  MoveL (T17595) to (111.78, 115.61, 18.9) mm, rotated rx 180 ry 0 rz -180 deg; joints [2.068, 71.073, -37.56, 3.741, -33.569, -3.119]
  Call Extruder 0.01417
  MoveL (T17596) to (111.39, 115.99, 18.9) mm, rotated rx 180 ry 0 rz -180 deg; joints [2.068, 71.073, -37.56, 3.741, -33.569, -3.119]
  Call Extruder 0.01304
  MoveL (T17597) to (110.9, 115.99, 18.9) mm, rotated rx 180 ry 0 rz -180 deg; joints [2.068, 71.073, -37.56, 3.741, -33.569, -3.119]
  Call Extruder 0.02638
  MoveL (T17598) to (111.61, 115.28, 18.9) mm, rotated rx 180 ry 0 rz -180 deg; joints [1.852, 70.394, -36.284, 3.299, -34.154, -2.731]
  Call Extruder 0.00969
  MoveL (T17599) to (111.44, 114.95, 18.9) mm, rotated rx 180 ry 0 rz -180 deg; joints [1.852, 70.394, -36.284, 3.299, -34.154, -2.731]
  Call Extruder 0.03859
  MoveL (T17600) to (110.4, 115.99, 18.9) mm, rotated rx 180 ry 0 rz -180 deg; joints [1.883, 70.309, -36.124, 3.349, -34.23, -2.77]
  Call Extruder 0.01304
  MoveL (T17601) to (109.91, 115.99, 18.9) mm, rotated rx 180 ry 0 rz -180 deg; joints [1.883, 70.309, -36.124, 3.349, -34.23, -2.77]
  Call Extruder 0.0508
  MoveL (T17602) to (111.27, 114.62, 18.9) mm, rotated rx 180 ry 0 rz -180 deg; joints [1.883, 70.309, -36.124, 3.349, -34.23, -2.77]
  Call Extruder 0.00969
  MoveL (T17603) to (111.11, 114.3, 18.9) mm, rotated rx 180 ry 0 rz -180 deg; joints [2.129, 71.08, -37.573, 3.852, -33.567, -3.211]
  Call Extruder 0.06301
  MoveL (T17604) to (109.41, 115.99, 18.9) mm, rotated rx 180 ry 0 rz -180 deg; joints [2.129, 71.08, -37.573, 3.852, -33.567, -3.211]
  Call Extruder 0.01304
  MoveL (T17605) to (108.91, 115.99, 18.9) mm, rotated rx 180 ry 0 rz -180 deg; joints [2.129, 71.08, -37.573, 3.852, -33.567, -3.211]
  Call Extruder 0.07523
  MoveL (T17606) to (110.94, 113.97, 18.9) mm, rotated rx 180 ry 0 rz -180 deg; joints [2.189, 71.086, -37.585, 3.962, -33.564, -3.303]
  Call Extruder 0.00969
  MoveL (T17607) to (110.77, 113.64, 18.9) mm, rotated rx 180 ry 0 rz -180 deg; joints [2.189, 71.086, -37.585, 3.962, -33.564, -3.303]
  Call Extruder 0.09322
  MoveL (T17608) to (108.26, 116.15, 18.9) mm, rotated rx 180 ry 0 rz -180 deg; joints [1.915, 70.224, -35.965, 3.398, -34.306, -2.808]
  Set speed (45.0 mm/s)
  Call Extruder -1.6
  MoveL (T17609) to (108.26, 116.15, 18.9) mm, rotated rx 180 ry 0 rz -180 deg; joints [1.915, 70.224, -35.965, 3.398, -34.306, -2.808]
  Set speed (120.0 mm/s)
  MoveL (T17610) to (108.26, 116.15, 18.9) mm, rotated rx 180 ry 0 rz -180 deg; joints [1.946, 70.14, -35.807, 3.448, -34.382, -2.847]
  Call Extruder -0.38
  MoveL (T17611) to (109.02, 115.39, 18.9) mm, rotated rx 180 ry 0 rz -180 deg; joints [1.946, 70.14, -35.807, 3.448, -34.382, -2.847]
  Set speed (45.0 mm/s)
  Call Extruder -0.02
  MoveL (T17612) to (109.02, 115.39, 18.9) mm, rotated rx 180 ry 0 rz -180 deg; joints [2.25, 71.093, -37.599, 4.072, -33.562, -3.395]
  Set speed (150.0 mm/s)
  MoveL (T17613) to (109.02, 115.39, 20.9) mm, rotated rx 180 ry 0 rz -180 deg; joints [2.25, 71.093, -37.599, 4.072, -33.562, -3.395]
  MoveL (T17614) to (107.75, 120.63, 20.9) mm, rotated rx 180 ry 0 rz -180 deg; joints [2.25, 71.093, -37.599, 4.072, -33.562, -3.395]
  MoveL (T17615) to (107.75, 120.63, 18.9) mm, rotated rx 180 ry 0 rz -180 deg; joints [2.311, 71.101, -37.612, 4.183, -33.559, -3.487]
  Set speed (40.0 mm/s)
  Call Extruder 2.0
  MoveL (T17616) to (107.75, 120.63, 18.9) mm, rotated rx 180 ry 0 rz -180 deg; joints [2.311, 71.101, -37.612, 4.183, -33.559, -3.487]
  Set speed (25.0 mm/s)
  MoveL (T17617) to (107.75, 120.63, 18.9) mm, rotated rx 180 ry 0 rz -180 deg; joints [2.311, 71.101, -37.612, 4.183, -33.559, -3.487]
  Call Extruder 0.0206
  MoveL (T17618) to (107.19, 121.19, 18.9) mm, rotated rx 180 ry 0 rz -180 deg; joints [1.978, 70.056, -35.649, 3.497, -34.457, -2.885]
  Call Extruder 0.01304
  MoveL (T17619) to (106.7, 121.19, 18.9) mm, rotated rx 180 ry 0 rz -180 deg; joints [1.978, 70.056, -35.649, 3.497, -34.457, -2.885]
  Call Extruder 0.03325
  MoveL (T17620) to (107.59, 120.29, 18.9) mm, rotated rx 180 ry 0 rz -180 deg; joints [2.009, 69.973, -35.492, 3.546, -34.532, -2.923]
  Call Extruder 0.01304
  MoveL (T17621) to (107.59, 119.8, 18.9) mm, rotated rx 180 ry 0 rz -180 deg; joints [2.009, 69.973, -35.492, 3.546, -34.532, -2.923]
  Call Extruder 0.0517
  MoveL (T17622) to (106.2, 121.19, 18.9) mm, rotated rx 180 ry 0 rz -180 deg; joints [2.009, 69.973, -35.492, 3.546, -34.532, -2.923]
  Call Extruder 0.01304
  MoveL (T17623) to (105.7, 121.19, 18.9) mm, rotated rx 180 ry 0 rz -180 deg; joints [2.371, 71.108, -37.626, 4.293, -33.556, -3.58]
  Call Extruder 0.07014
  MoveL (T17624) to (107.59, 119.3, 18.9) mm, rotated rx 180 ry 0 rz -180 deg; joints [2.371, 71.108, -37.626, 4.293, -33.556, -3.58]
  Call Extruder 0.01304
  MoveL (T17625) to (107.59, 118.8, 18.9) mm, rotated rx 180 ry 0 rz -180 deg; joints [2.371, 71.108, -37.626, 4.293, -33.556, -3.58]
  Call Extruder 0.08858
  MoveL (T17626) to (105.21, 121.19, 18.9) mm, rotated rx 180 ry 0 rz -180 deg; joints [2.432, 71.116, -37.64, 4.403, -33.553, -3.672]
  Call Extruder 0.01304
  MoveL (T17627) to (104.71, 121.19, 18.9) mm, rotated rx 180 ry 0 rz -180 deg; joints [2.432, 71.116, -37.64, 4.403, -33.553, -3.672]
  Call Extruder 0.10702
  MoveL (T17628) to (107.59, 118.31, 18.9) mm, rotated rx 180 ry 0 rz -180 deg; joints [2.432, 71.116, -37.64, 4.403, -33.553, -3.672]
  Call Extruder 0.01304
  MoveL (T17629) to (107.59, 117.81, 18.9) mm, rotated rx 180 ry 0 rz -180 deg; joints [2.041, 69.89, -35.336, 3.595, -34.606, -2.961]
  Call Extruder 0.12546
  MoveL (T17630) to (104.22, 121.19, 18.9) mm, rotated rx 180 ry 0 rz -180 deg; joints [2.041, 69.89, -35.336, 3.595, -34.606, -2.961]
  Call Extruder 0.01054
  MoveL (T17631) to (103.81, 121.19, 18.9) mm, rotated rx 180 ry 0 rz -180 deg; joints [2.048, 69.871, -35.301, 3.606, -34.623, -2.969]
  Call Extruder 0.0025
  MoveL (T17632) to (103.81, 121.09, 18.9) mm, rotated rx 180 ry 0 rz -180 deg; joints [2.048, 69.871, -35.301, 3.606, -34.623, -2.969]
  Call Extruder 0.14037
  MoveL (T17633) to (107.59, 117.31, 18.9) mm, rotated rx 180 ry 0 rz -180 deg; joints [2.053, 69.865, -35.291, 3.615, -34.628, -2.976]
  Call Extruder 0.01304
  MoveL (T17634) to (107.59, 116.82, 18.9) mm, rotated rx 180 ry 0 rz -180 deg; joints [2.053, 69.865, -35.291, 3.615, -34.628, -2.976]
  Call Extruder 0.14037
  MoveL (T17635) to (103.81, 120.59, 18.9) mm, rotated rx 180 ry 0 rz -180 deg; joints [2.053, 69.865, -35.291, 3.615, -34.628, -2.976]
  Call Extruder 0.01304
  MoveL (T17636) to (103.81, 120.1, 18.9) mm, rotated rx 180 ry 0 rz -180 deg; joints [2.053, 69.865, -35.291, 3.615, -34.628, -2.976]
  Call Extruder 0.14037
  MoveL (T17637) to (107.59, 116.32, 18.9) mm, rotated rx 180 ry 0 rz -180 deg; joints [2.093, 69.869, -35.298, 3.686, -34.626, -3.034]
  Call Extruder 0.00862
  MoveL (T17638) to (107.59, 115.99, 18.9) mm, rotated rx 180 ry 0 rz -180 deg; joints [2.493, 71.124, -37.655, 4.514, -33.55, -3.764]
  Call Extruder 0.00862
  MoveL (T17639) to (107.92, 115.99, 18.9) mm, rotated rx 180 ry 0 rz -180 deg; joints [2.493, 71.124, -37.655, 4.514, -33.55, -3.764]
  Call Extruder 0.09965
  MoveL (T17640) to (110.6, 113.31, 18.9) mm, rotated rx 180 ry 0 rz -180 deg; joints [2.553, 71.132, -37.67, 4.624, -33.547, -3.856]
  Call Extruder 0.00969
  MoveL (T17641) to (110.44, 112.98, 18.9) mm, rotated rx 180 ry 0 rz -180 deg; joints [2.553, 71.132, -37.67, 4.624, -33.547, -3.856]
  Call Extruder 0.24597
  MoveL (T17642) to (103.81, 119.6, 18.9) mm, rotated rx 180 ry 0 rz -180 deg; joints [2.553, 71.132, -37.67, 4.624, -33.547, -3.856]
  Call Extruder 0.01304
  MoveL (T17643) to (103.81, 119.11, 18.9) mm, rotated rx 180 ry 0 rz -180 deg; joints [2.154, 69.876, -35.31, 3.794, -34.624, -3.123]
  Call Extruder 0.23974
  MoveL (T17644) to (110.27, 112.65, 18.9) mm, rotated rx 180 ry 0 rz -180 deg; joints [2.154, 69.876, -35.31, 3.794, -34.624, -3.123]
  Call Extruder 0.00969
  MoveL (T17645) to (110.1, 112.32, 18.9) mm, rotated rx 180 ry 0 rz -180 deg; joints [2.154, 69.876, -35.31, 3.794, -34.624, -3.123]
  Call Extruder 0.23351
  MoveL (T17646) to (103.81, 118.61, 18.9) mm, rotated rx 180 ry 0 rz -180 deg; joints [2.216, 69.882, -35.322, 3.902, -34.622, -3.212]
  Call Extruder 0.01304
  MoveL (T17647) to (103.81, 118.11, 18.9) mm, rotated rx 180 ry 0 rz -180 deg; joints [2.216, 69.882, -35.322, 3.902, -34.622, -3.212]
  Call Extruder 0.22728
  MoveL (T17648) to (109.93, 111.99, 18.9) mm, rotated rx 180 ry 0 rz -180 deg; joints [2.614, 71.14, -37.686, 4.734, -33.544, -3.949]
  Call Extruder 0.00969
  MoveL (T17649) to (109.76, 111.67, 18.9) mm, rotated rx 180 ry 0 rz -180 deg; joints [2.614, 71.14, -37.686, 4.734, -33.544, -3.949]
  Call Extruder 0.22105
  MoveL (T17650) to (103.81, 117.62, 18.9) mm, rotated rx 180 ry 0 rz -180 deg; joints [2.675, 71.148, -37.701, 4.845, -33.541, -4.041]
  Call Extruder 0.01304
  MoveL (T17651) to (103.81, 117.12, 18.9) mm, rotated rx 180 ry 0 rz -180 deg; joints [2.675, 71.148, -37.701, 4.845, -33.541, -4.041]
  Call Extruder 0.21482
  MoveL (T17652) to (109.6, 111.34, 18.9) mm, rotated rx 180 ry 0 rz -180 deg; joints [2.675, 71.148, -37.701, 4.845, -33.541, -4.041]
  Call Extruder 0.00969
  MoveL (T17653) to (109.43, 111.01, 18.9) mm, rotated rx 180 ry 0 rz -180 deg; joints [2.277, 69.889, -35.335, 4.01, -34.62, -3.302]
  Call Extruder 0.2086
  MoveL (T17654) to (103.81, 116.62, 18.9) mm, rotated rx 180 ry 0 rz -180 deg; joints [2.277, 69.889, -35.335, 4.01, -34.62, -3.302]
  Call Extruder 0.01304
  MoveL (T17655) to (103.81, 116.13, 18.9) mm, rotated rx 180 ry 0 rz -180 deg; joints [2.338, 69.896, -35.348, 4.118, -34.617, -3.391]
  Call Extruder 0.20237
  MoveL (T17656) to (109.26, 110.68, 18.9) mm, rotated rx 180 ry 0 rz -180 deg; joints [2.338, 69.896, -35.348, 4.118, -34.617, -3.391]
  Call Extruder 0.00969
  MoveL (T17657) to (109.09, 110.35, 18.9) mm, rotated rx 180 ry 0 rz -180 deg; joints [2.71, 71.074, -37.561, 4.9, -33.609, -4.084]
  Call Extruder 0.19614
  MoveL (T17658) to (103.81, 115.63, 18.9) mm, rotated rx 180 ry 0 rz -180 deg; joints [2.713, 70.893, -37.222, 4.885, -33.767, -4.064]
  Call Extruder 0.01304
  MoveL (T17659) to (103.81, 115.13, 18.9) mm, rotated rx 180 ry 0 rz -180 deg; joints [2.713, 70.893, -37.222, 4.885, -33.767, -4.064]
  Call Extruder 0.18991
  MoveL (T17660) to (108.93, 110.02, 18.9) mm, rotated rx 180 ry 0 rz -180 deg; joints [2.399, 69.903, -35.361, 4.226, -34.615, -3.48]
  Call Extruder 0.00969
  MoveL (T17661) to (108.76, 109.69, 18.9) mm, rotated rx 180 ry 0 rz -180 deg; joints [2.399, 69.903, -35.361, 4.226, -34.615, -3.48]
  Call Extruder 0.18368
  MoveL (T17662) to (103.81, 114.64, 18.9) mm, rotated rx 180 ry 0 rz -180 deg; joints [2.399, 69.903, -35.361, 4.226, -34.615, -3.48]
  Call Extruder 0.01304
  MoveL (T17663) to (103.81, 114.14, 18.9) mm, rotated rx 180 ry 0 rz -180 deg; joints [2.46, 69.91, -35.374, 4.334, -34.612, -3.569]
  Call Extruder 0.17745
  MoveL (T17664) to (108.59, 109.36, 18.9) mm, rotated rx 180 ry 0 rz -180 deg; joints [2.46, 69.91, -35.374, 4.334, -34.612, -3.569]
  Call Extruder 0.00969
  MoveL (T17665) to (108.42, 109.04, 18.9) mm, rotated rx 180 ry 0 rz -180 deg; joints [2.716, 70.714, -36.886, 4.87, -33.924, -4.044]
  Call Extruder 0.17122
  MoveL (T17666) to (103.81, 113.64, 18.9) mm, rotated rx 180 ry 0 rz -180 deg; joints [2.716, 70.714, -36.886, 4.87, -33.924, -4.044]
  Call Extruder 0.01304
  MoveL (T17667) to (103.81, 113.15, 18.9) mm, rotated rx 180 ry 0 rz -180 deg; joints [2.716, 70.714, -36.886, 4.87, -33.924, -4.044]
  Call Extruder 0.16499
  MoveL (T17668) to (108.25, 108.71, 18.9) mm, rotated rx 180 ry 0 rz -180 deg; joints [2.719, 70.545, -36.568, 4.857, -34.073, -4.026]
  Call Extruder 0.00969
  MoveL (T17669) to (108.09, 108.38, 18.9) mm, rotated rx 180 ry 0 rz -180 deg; joints [2.719, 70.545, -36.568, 4.857, -34.073, -4.026]
  Call Extruder 0.15876
  MoveL (T17670) to (103.81, 112.65, 18.9) mm, rotated rx 180 ry 0 rz -180 deg; joints [2.717, 70.53, -36.539, 4.852, -34.086, -4.021]
  Call Extruder 0.01304
  MoveL (T17671) to (103.81, 112.16, 18.9) mm, rotated rx 180 ry 0 rz -180 deg; joints [2.503, 69.861, -35.282, 4.404, -34.658, -3.625]
  Call Extruder 0.15253
  MoveL (T17672) to (107.92, 108.05, 18.9) mm, rotated rx 180 ry 0 rz -180 deg; joints [2.503, 69.861, -35.282, 4.404, -34.658, -3.625]
  Call Extruder 0.00969
  MoveL (T17673) to (107.75, 107.72, 18.9) mm, rotated rx 180 ry 0 rz -180 deg; joints [2.503, 69.861, -35.282, 4.404, -34.658, -3.625]
  Call Extruder 0.1463
  MoveL (T17674) to (103.81, 111.66, 18.9) mm, rotated rx 180 ry 0 rz -180 deg; joints [2.503, 69.861, -35.282, 4.404, -34.658, -3.625]
  Call Extruder 0.01304
  MoveL (T17675) to (103.81, 111.16, 18.9) mm, rotated rx 180 ry 0 rz -180 deg; joints [2.503, 69.861, -35.282, 4.404, -34.658, -3.625]
  Call Extruder 0.14007
  MoveL (T17676) to (107.58, 107.39, 18.9) mm, rotated rx 180 ry 0 rz -180 deg; joints [2.503, 69.861, -35.282, 4.404, -34.658, -3.625]
  Call Extruder 0.00439
  MoveL (T17677) to (107.51, 107.24, 18.9) mm, rotated rx 180 ry 0 rz -180 deg; joints [2.503, 69.861, -35.282, 4.404, -34.658, -3.625]
  Call Extruder 0.00713
  MoveL (T17678) to (107.51, 106.97, 18.9) mm, rotated rx 180 ry 0 rz -180 deg; joints [2.503, 69.861, -35.282, 4.404, -34.658, -3.625]
  Call Extruder 0.13724
  MoveL (T17679) to (103.81, 110.67, 18.9) mm, rotated rx 180 ry 0 rz -180 deg; joints [2.503, 69.861, -35.282, 4.404, -34.658, -3.625]
  Call Extruder 0.01304
  MoveL (T17680) to (103.81, 110.17, 18.9) mm, rotated rx 180 ry 0 rz -180 deg; joints [2.503, 69.861, -35.282, 4.404, -34.658, -3.625]
  Call Extruder 0.13724
  MoveL (T17681) to (107.51, 106.47, 18.9) mm, rotated rx 180 ry 0 rz -180 deg; joints [2.579, 70.095, -35.723, 4.561, -34.457, -3.763]
  Call Extruder 0.01304
  MoveL (T17682) to (107.51, 105.98, 18.9) mm, rotated rx 180 ry 0 rz -180 deg; joints [2.579, 70.095, -35.723, 4.561, -34.457, -3.763]
  Call Extruder 0.13724
  MoveL (T17683) to (103.81, 109.67, 18.9) mm, rotated rx 180 ry 0 rz -180 deg; joints [2.579, 70.095, -35.723, 4.561, -34.457, -3.763]
  Call Extruder 0.01304
  MoveL (T17684) to (103.81, 109.18, 18.9) mm, rotated rx 180 ry 0 rz -180 deg; joints [2.579, 70.095, -35.723, 4.561, -34.457, -3.763]
  Call Extruder 0.13724
  MoveL (T17685) to (107.51, 105.48, 18.9) mm, rotated rx 180 ry 0 rz -180 deg; joints [2.579, 70.095, -35.723, 4.561, -34.457, -3.763]
  Call Extruder 0.01304
  MoveL (T17686) to (107.51, 104.99, 18.9) mm, rotated rx 180 ry 0 rz -180 deg; joints [2.579, 70.095, -35.723, 4.561, -34.457, -3.763]
  Call Extruder 0.13724
  MoveL (T17687) to (103.81, 108.68, 18.9) mm, rotated rx 180 ry 0 rz -180 deg; joints [2.579, 70.095, -35.723, 4.561, -34.457, -3.763]
  Call Extruder 0.01304
  MoveL (T17688) to (103.81, 108.18, 18.9) mm, rotated rx 180 ry 0 rz -180 deg; joints [1.869, 68.982, -34.029, 3.26, -34.996, -2.671]
  Call Extruder 0.13724
  MoveL (T17689) to (107.51, 104.49, 18.9) mm, rotated rx 180 ry 0 rz -180 deg; joints [1.869, 69.215, -34.069, 3.244, -35.189, -2.652]
  Call Extruder 0.01304
  MoveL (T17690) to (107.51, 103.99, 18.9) mm, rotated rx 180 ry 0 rz -180 deg; joints [1.869, 69.215, -34.069, 3.244, -35.189, -2.652]
  Call Extruder 0.13724
  MoveL (T17691) to (103.81, 107.69, 18.9) mm, rotated rx 180 ry 0 rz -180 deg; joints [1.869, 69.215, -34.069, 3.244, -35.189, -2.652]
  Call Extruder 0.01304
  MoveL (T17692) to (103.81, 107.19, 18.9) mm, rotated rx 180 ry 0 rz -180 deg; joints [1.869, 69.215, -34.069, 3.244, -35.189, -2.652]
  Call Extruder 0.12546
  MoveL (T17693) to (107.19, 103.81, 18.9) mm, rotated rx 180 ry 0 rz -180 deg; joints [1.869, 69.215, -34.069, 3.244, -35.189, -2.652]
  Call Extruder 0.01304
  MoveL (T17694) to (106.69, 103.81, 18.9) mm, rotated rx 180 ry 0 rz -180 deg; joints [1.869, 69.215, -34.069, 3.244, -35.189, -2.652]
  Call Extruder 0.10702
  MoveL (T17695) to (103.81, 106.69, 18.9) mm, rotated rx 180 ry 0 rz -180 deg; joints [1.869, 69.215, -34.069, 3.244, -35.189, -2.652]
  Call Extruder 0.01304
  MoveL (T17696) to (103.81, 106.2, 18.9) mm, rotated rx 180 ry 0 rz -180 deg; joints [1.869, 69.215, -34.069, 3.244, -35.189, -2.652]
  Call Extruder 0.08857
  MoveL (T17697) to (106.2, 103.81, 18.9) mm, rotated rx 180 ry 0 rz -180 deg; joints [1.869, 69.215, -34.069, 3.244, -35.189, -2.652]
  Call Extruder 0.01304
  MoveL (T17698) to (105.7, 103.81, 18.9) mm, rotated rx 180 ry 0 rz -180 deg; joints [1.874, 68.78, -33.251, 3.223, -35.572, -2.622]
  Call Extruder 0.07013
  MoveL (T17699) to (103.81, 105.7, 18.9) mm, rotated rx 180 ry 0 rz -180 deg; joints [1.874, 68.78, -33.251, 3.223, -35.572, -2.622]
  Call Extruder 0.01304
  MoveL (T17700) to (103.81, 105.2, 18.9) mm, rotated rx 180 ry 0 rz -180 deg; joints [1.866, 68.722, -33.142, 3.205, -35.622, -2.606]
  Call Extruder 0.05169
  MoveL (T17701) to (105.2, 103.81, 18.9) mm, rotated rx 180 ry 0 rz -180 deg; joints [1.866, 68.722, -33.142, 3.205, -35.622, -2.606]
  Call Extruder 0.01304
  MoveL (T17702) to (104.71, 103.81, 18.9) mm, rotated rx 180 ry 0 rz -180 deg; joints [1.866, 68.722, -33.142, 3.205, -35.622, -2.606]
  Call Extruder 0.03325
  MoveL (T17703) to (103.81, 104.71, 18.9) mm, rotated rx 180 ry 0 rz -180 deg; joints [1.866, 68.722, -33.142, 3.205, -35.622, -2.606]
  Call Extruder 0.01304
  MoveL (T17704) to (103.81, 104.21, 18.9) mm, rotated rx 180 ry 0 rz -180 deg; joints [1.866, 68.722, -33.142, 3.205, -35.622, -2.606]
  Call Extruder 0.02059
  MoveL (T17705) to (104.37, 103.66, 18.9) mm, rotated rx 180 ry 0 rz -180 deg; joints [2.818, 66.261, -28.52, 4.598, -37.83, -3.634]
  Set speed (45.0 mm/s)
  Call Extruder -1.6
  MoveL (T17706) to (104.37, 103.66, 18.9) mm, rotated rx 180 ry 0 rz -180 deg; joints [2.818, 66.261, -28.52, 4.598, -37.83, -3.634]
  Set speed (120.0 mm/s)
  MoveL (T17707) to (104.37, 103.66, 18.9) mm, rotated rx 180 ry 0 rz -180 deg; joints [2.938, 66.275, -28.547, 4.795, -37.825, -3.791]
  Call Extruder -0.27925
  MoveL (T17708) to (103.81, 104.21, 18.9) mm, rotated rx 180 ry 0 rz -180 deg; joints [2.938, 66.275, -28.547, 4.795, -37.825, -3.791]
  Call Extruder -0.10075
  MoveL (T17709) to (103.81, 104.5, 18.9) mm, rotated rx 180 ry 0 rz -180 deg; joints [2.938, 66.275, -28.547, 4.795, -37.825, -3.791]
  Set speed (45.0 mm/s)
  Call Extruder -0.02
  MoveL (T17710) to (103.81, 104.5, 18.9) mm, rotated rx 180 ry 0 rz -180 deg; joints [3.295, 67.241, -30.36, 5.479, -37.007, -4.38]
  Set speed (150.0 mm/s)
  MoveL (T17711) to (103.81, 104.5, 20.9) mm, rotated rx 180 ry 0 rz -180 deg; joints [3.295, 67.241, -30.36, 5.479, -37.007, -4.38]
  MoveL (T17712) to (117.55, 120.5, 20.9) mm, rotated rx 180 ry 0 rz -180 deg; joints [3.288, 67.539, -30.92, 5.501, -36.745, -4.413]
  MoveL (T17713) to (117.55, 120.5, 18.9) mm, rotated rx 180 ry 0 rz -180 deg; joints [3.288, 67.539, -30.92, 5.501, -36.745, -4.413]
  Set speed (40.0 mm/s)
  Call Extruder 2.0
  MoveL (T17714) to (117.55, 120.5, 18.9) mm, rotated rx 180 ry 0 rz -180 deg; joints [2.356, 69.777, -35.125, 4.138, -34.722, -3.403]
  Call Extruder 0.02915
  MoveL (T17715) to (116.89, 121.16, 18.9) mm, rotated rx 180 ry 0 rz -180 deg; joints [2.356, 69.777, -35.125, 4.138, -34.722, -3.403]
  Call Extruder 0.0184
  MoveL (T17716) to (116.3, 121.16, 18.9) mm, rotated rx 180 ry 0 rz -180 deg; joints [2.356, 69.777, -35.125, 4.138, -34.722, -3.403]
  Call Extruder 0.04381
  MoveL (T17717) to (117.29, 120.16, 18.9) mm, rotated rx 180 ry 0 rz -180 deg; joints [2.29, 69.769, -35.111, 4.022, -34.725, -3.308]
  Call Extruder 0.0184
  MoveL (T17718) to (116.7, 120.16, 18.9) mm, rotated rx 180 ry 0 rz -180 deg; joints [2.29, 69.769, -35.111, 4.022, -34.725, -3.308]
  Call Extruder 0.04381
  MoveL (T17719) to (115.71, 121.16, 18.9) mm, rotated rx 180 ry 0 rz -180 deg; joints [2.29, 69.769, -35.111, 4.022, -34.725, -3.308]
  Call Extruder 0.0184
  MoveL (T17720) to (115.12, 121.16, 18.9) mm, rotated rx 180 ry 0 rz -180 deg; joints [1.775, 68.278, -32.309, 3.02, -36.007, -2.444]
  Call Extruder 0.04381
  MoveL (T17721) to (116.11, 120.16, 18.9) mm, rotated rx 180 ry 0 rz -180 deg; joints [1.775, 68.278, -32.309, 3.02, -36.007, -2.444]
  Call Extruder 0.0184
  MoveL (T17722) to (115.52, 120.16, 18.9) mm, rotated rx 180 ry 0 rz -180 deg; joints [1.875, 68.036, -31.854, 3.173, -36.224, -2.561]
  Call Extruder 0.04381
  MoveL (T17723) to (114.53, 121.16, 18.9) mm, rotated rx 180 ry 0 rz -180 deg; joints [1.875, 68.036, -31.854, 3.173, -36.224, -2.561]
  Call Extruder 0.0184
  MoveL (T17724) to (113.94, 121.16, 18.9) mm, rotated rx 180 ry 0 rz -180 deg; joints [1.875, 68.036, -31.854, 3.173, -36.224, -2.561]
  Call Extruder 0.04381
  MoveL (T17725) to (114.93, 120.16, 18.9) mm, rotated rx 180 ry 0 rz -180 deg; joints [1.884, 67.982, -31.752, 3.186, -36.272, -2.569]
  Call Extruder 0.0184
  MoveL (T17726) to (114.34, 120.16, 18.9) mm, rotated rx 180 ry 0 rz -180 deg; joints [1.884, 67.982, -31.752, 3.186, -36.272, -2.569]
  Call Extruder 0.04381
  MoveL (T17727) to (113.35, 121.16, 18.9) mm, rotated rx 180 ry 0 rz -180 deg; joints [1.884, 67.982, -31.752, 3.186, -36.272, -2.569]
  Call Extruder 0.0184
  MoveL (T17728) to (112.76, 121.16, 18.9) mm, rotated rx 180 ry 0 rz -180 deg; joints [1.888, 67.723, -31.266, 3.174, -36.499, -2.553]
  Call Extruder 0.04381
  MoveL (T17729) to (113.75, 120.16, 18.9) mm, rotated rx 180 ry 0 rz -180 deg; joints [1.888, 67.723, -31.266, 3.174, -36.499, -2.553]
  Call Extruder 0.0184
  MoveL (T17730) to (113.16, 120.16, 18.9) mm, rotated rx 180 ry 0 rz -180 deg; joints [1.888, 67.723, -31.266, 3.174, -36.499, -2.553]
  Call Extruder 0.04381
  MoveL (T17731) to (112.17, 121.16, 18.9) mm, rotated rx 180 ry 0 rz -180 deg; joints [1.888, 67.723, -31.266, 3.174, -36.499, -2.553]
  Call Extruder 0.0184
  MoveL (T17732) to (111.58, 121.16, 18.9) mm, rotated rx 180 ry 0 rz -180 deg; joints [1.888, 67.723, -31.266, 3.174, -36.499, -2.553]
  Call Extruder 0.04381
  MoveL (T17733) to (112.57, 120.16, 18.9) mm, rotated rx 180 ry 0 rz -180 deg; joints [1.888, 67.723, -31.266, 3.174, -36.499, -2.553]
  Call Extruder 0.0184
  MoveL (T17734) to (111.98, 120.16, 18.9) mm, rotated rx 180 ry 0 rz -180 deg; joints [1.888, 67.723, -31.266, 3.174, -36.499, -2.553]
  Call Extruder 0.04381
  MoveL (T17735) to (110.99, 121.16, 18.9) mm, rotated rx 180 ry 0 rz -180 deg; joints [1.888, 67.723, -31.266, 3.174, -36.499, -2.553]
  Call Extruder 0.0184
  MoveL (T17736) to (110.4, 121.16, 18.9) mm, rotated rx 180 ry 0 rz -180 deg; joints [1.888, 67.723, -31.266, 3.174, -36.499, -2.553]
  Call Extruder 0.04381
  MoveL (T17737) to (111.39, 120.16, 18.9) mm, rotated rx 180 ry 0 rz -180 deg; joints [1.884, 67.982, -31.752, 3.186, -36.272, -2.569]
  Call Extruder 0.0184
  MoveL (T17738) to (110.81, 120.16, 18.9) mm, rotated rx 180 ry 0 rz -180 deg; joints [1.884, 67.982, -31.752, 3.186, -36.272, -2.569]
  Call Extruder 0.04381
  MoveL (T17739) to (109.81, 121.16, 18.9) mm, rotated rx 180 ry 0 rz -180 deg; joints [1.884, 67.982, -31.752, 3.186, -36.272, -2.569]
  Call Extruder 0.0184
  MoveL (T17740) to (109.22, 121.16, 18.9) mm, rotated rx 180 ry 0 rz -180 deg; joints [1.879, 68.012, -31.808, 3.179, -36.245, -2.565]
  Call Extruder 0.04381
  MoveL (T17741) to (110.22, 120.16, 18.9) mm, rotated rx 180 ry 0 rz -180 deg; joints [1.879, 68.012, -31.808, 3.179, -36.245, -2.565]
  Call Extruder 0.0184
  MoveL (T17742) to (109.62, 120.16, 18.9) mm, rotated rx 180 ry 0 rz -180 deg; joints [1.879, 68.012, -31.808, 3.179, -36.245, -2.565]
  Call Extruder 0.04381
  MoveL (T17743) to (108.63, 121.16, 18.9) mm, rotated rx 180 ry 0 rz -180 deg; joints [1.879, 68.012, -31.808, 3.179, -36.245, -2.565]
  Call Extruder 0.0184
  MoveL (T17744) to (108.04, 121.16, 18.9) mm, rotated rx 180 ry 0 rz -180 deg; joints [1.879, 68.012, -31.808, 3.179, -36.245, -2.565]
  Call Extruder 0.04381
  MoveL (T17745) to (109.04, 120.16, 18.9) mm, rotated rx 180 ry 0 rz -180 deg; joints [1.879, 68.012, -31.808, 3.179, -36.245, -2.565]
  Call Extruder 0.0184
  MoveL (T17746) to (108.45, 120.16, 18.9) mm, rotated rx 180 ry 0 rz -180 deg; joints [1.879, 68.012, -31.808, 3.179, -36.245, -2.565]
  Call Extruder 0.02914
  MoveL (T17747) to (107.79, 120.82, 18.9) mm, rotated rx 180 ry 0 rz -180 deg; joints [1.879, 68.012, -31.808, 3.179, -36.245, -2.565]
  Set speed (45.0 mm/s)
  Call Extruder -1.6
  MoveL (T17748) to (107.79, 120.82, 18.9) mm, rotated rx 180 ry 0 rz -180 deg; joints [1.476, 70.512, -36.902, 2.665, -33.639, -2.219]
  Set speed (120.0 mm/s)
  MoveL (T17749) to (107.79, 120.82, 18.9) mm, rotated rx 180 ry 0 rz -180 deg; joints [1.476, 70.745, -36.944, 2.652, -33.83, -2.203]
  Call Extruder -0.33277
  MoveL (T17750) to (108.45, 120.16, 18.9) mm, rotated rx 180 ry 0 rz -180 deg; joints [1.476, 70.745, -36.944, 2.652, -33.83, -2.203]
  Call Extruder -0.04723
  MoveL (T17751) to (108.58, 120.16, 18.9) mm, rotated rx 180 ry 0 rz -180 deg; joints [1.476, 70.745, -36.944, 2.652, -33.83, -2.203]
  Set speed (45.0 mm/s)
  Call Extruder -0.02
  MoveL (T17752) to (108.58, 120.16, 18.9) mm, rotated rx 180 ry 0 rz -180 deg; joints [1.476, 70.745, -36.944, 2.652, -33.83, -2.203]
  Set speed (150.0 mm/s)
  MoveL (T17753) to (108.58, 120.16, 20.9) mm, rotated rx 180 ry 0 rz -180 deg; joints [1.476, 70.745, -36.944, 2.652, -33.83, -2.203]
  MoveL (T17754) to (121.34, 120.63, 20.9) mm, rotated rx 180 ry 0 rz -180 deg; joints [1.476, 70.745, -36.944, 2.652, -33.83, -2.203]
  MoveL (T17755) to (121.34, 120.63, 18.9) mm, rotated rx 180 ry 0 rz -180 deg; joints [1.476, 70.745, -36.944, 2.652, -33.83, -2.203]
  Set speed (40.0 mm/s)
  Call Extruder 2.0
  MoveL (T17756) to (121.34, 120.63, 18.9) mm, rotated rx 180 ry 0 rz -180 deg; joints [1.476, 70.745, -36.944, 2.652, -33.83, -2.203]
  Set speed (25.0 mm/s)
  MoveL (T17757) to (121.34, 120.63, 18.9) mm, rotated rx 180 ry 0 rz -180 deg; joints [1.476, 70.745, -36.944, 2.652, -33.83, -2.203]
  Call Extruder 0.02055
  MoveL (T17758) to (120.79, 121.19, 18.9) mm, rotated rx 180 ry 0 rz -180 deg; joints [1.4, 70.513, -36.507, 2.502, -34.031, -2.074]
  Call Extruder 0.01301
  MoveL (T17759) to (120.29, 121.19, 18.9) mm, rotated rx 180 ry 0 rz -180 deg; joints [1.4, 70.513, -36.507, 2.502, -34.031, -2.074]
  Call Extruder 0.03317
  MoveL (T17760) to (121.19, 120.29, 18.9) mm, rotated rx 180 ry 0 rz -180 deg; joints [1.402, 70.332, -36.168, 2.495, -34.19, -2.064]
  Call Extruder 0.01301
  MoveL (T17761) to (121.19, 119.8, 18.9) mm, rotated rx 180 ry 0 rz -180 deg; joints [1.402, 70.332, -36.168, 2.495, -34.19, -2.064]
  Call Extruder 0.05158
  MoveL (T17762) to (119.8, 121.19, 18.9) mm, rotated rx 180 ry 0 rz -180 deg; joints [1.402, 70.332, -36.168, 2.495, -34.19, -2.064]
  Call Extruder 0.01301
  MoveL (T17763) to (119.3, 121.19, 18.9) mm, rotated rx 180 ry 0 rz -180 deg; joints [1.402, 70.332, -36.168, 2.495, -34.19, -2.064]
  Call Extruder 0.06998
  MoveL (T17764) to (121.19, 119.3, 18.9) mm, rotated rx 180 ry 0 rz -180 deg; joints [1.52, 70.692, -36.843, 2.727, -33.878, -2.264]
  Call Extruder 0.01301
  MoveL (T17765) to (121.19, 118.81, 18.9) mm, rotated rx 180 ry 0 rz -180 deg; joints [1.52, 70.692, -36.843, 2.727, -33.878, -2.264]
  Call Extruder 0.08838
  MoveL (T17766) to (118.81, 121.19, 18.9) mm, rotated rx 180 ry 0 rz -180 deg; joints [1.582, 70.696, -36.853, 2.839, -33.876, -2.357]
  Call Extruder 0.01301
  MoveL (T17767) to (118.31, 121.19, 18.9) mm, rotated rx 180 ry 0 rz -180 deg; joints [1.582, 70.696, -36.853, 2.839, -33.876, -2.357]
  Call Extruder 0.10679
  MoveL (T17768) to (121.19, 118.31, 18.9) mm, rotated rx 180 ry 0 rz -180 deg; joints [1.403, 70.153, -35.831, 2.488, -34.347, -2.054]
  Call Extruder 0.01301
  MoveL (T17769) to (121.19, 117.81, 18.9) mm, rotated rx 180 ry 0 rz -180 deg; joints [1.403, 70.153, -35.831, 2.488, -34.347, -2.054]
  Call Extruder 0.12519
  MoveL (T17770) to (117.81, 121.19, 18.9) mm, rotated rx 180 ry 0 rz -180 deg; joints [1.403, 70.153, -35.831, 2.488, -34.347, -2.054]
  Call Extruder 0.00188
  MoveL (T17771) to (117.74, 121.19, 18.9) mm, rotated rx 180 ry 0 rz -180 deg; joints [1.405, 69.975, -35.497, 2.48, -34.503, -2.044]
  Call Extruder 0.01114
  MoveL (T17772) to (117.74, 120.76, 18.9) mm, rotated rx 180 ry 0 rz -180 deg; joints [1.405, 69.975, -35.497, 2.48, -34.503, -2.044]
  Call Extruder 0.12784
  MoveL (T17773) to (121.19, 117.32, 18.9) mm, rotated rx 180 ry 0 rz -180 deg; joints [1.624, 70.639, -36.744, 2.91, -33.929, -2.415]
  Call Extruder 0.01301
  MoveL (T17774) to (121.19, 116.82, 18.9) mm, rotated rx 180 ry 0 rz -180 deg; joints [1.624, 70.639, -36.744, 2.91, -33.929, -2.415]
  Call Extruder 0.12784
  MoveL (T17775) to (117.74, 120.27, 18.9) mm, rotated rx 180 ry 0 rz -180 deg; joints [1.656, 70.55, -36.578, 2.962, -34.008, -2.456]
  Call Extruder 0.01301
  MoveL (T17776) to (117.74, 119.77, 18.9) mm, rotated rx 180 ry 0 rz -180 deg; joints [1.656, 70.55, -36.578, 2.962, -34.008, -2.456]
  Call Extruder 0.12784
  MoveL (T17777) to (121.19, 116.33, 18.9) mm, rotated rx 180 ry 0 rz -180 deg; joints [1.406, 69.799, -35.166, 2.473, -34.658, -2.035]
  Call Extruder 0.01301
  MoveL (T17778) to (121.19, 115.83, 18.9) mm, rotated rx 180 ry 0 rz -180 deg; joints [1.406, 69.799, -35.166, 2.473, -34.658, -2.035]
  Call Extruder 0.12784
  MoveL (T17779) to (117.74, 119.27, 18.9) mm, rotated rx 180 ry 0 rz -180 deg; joints [1.406, 69.799, -35.166, 2.473, -34.658, -2.035]
  Call Extruder 0.01301
  MoveL (T17780) to (117.74, 118.78, 18.9) mm, rotated rx 180 ry 0 rz -180 deg; joints [1.408, 69.624, -34.837, 2.466, -34.812, -2.025]
  Call Extruder 0.12784
  MoveL (T17781) to (121.19, 115.33, 18.9) mm, rotated rx 180 ry 0 rz -180 deg; joints [1.408, 69.624, -34.837, 2.466, -34.812, -2.025]
  Call Extruder 0.01301
  MoveL (T17782) to (121.19, 114.84, 18.9) mm, rotated rx 180 ry 0 rz -180 deg; joints [1.408, 69.624, -34.837, 2.466, -34.812, -2.025]
  Call Extruder 0.12784
  MoveL (T17783) to (117.74, 118.28, 18.9) mm, rotated rx 180 ry 0 rz -180 deg; joints [1.408, 69.624, -34.837, 2.466, -34.812, -2.025]
  Call Extruder 0.00527
  MoveL (T17784) to (117.74, 118.08, 18.9) mm, rotated rx 180 ry 0 rz -180 deg; joints [1.688, 70.462, -36.412, 3.013, -34.087, -2.496]
  Call Extruder 0.00575
  MoveL (T17785) to (117.64, 117.89, 18.9) mm, rotated rx 180 ry 0 rz -180 deg; joints [1.688, 70.462, -36.412, 3.013, -34.087, -2.496]
  Call Extruder 0.13155
  MoveL (T17786) to (121.19, 114.34, 18.9) mm, rotated rx 180 ry 0 rz -180 deg; joints [1.72, 70.375, -36.248, 3.064, -34.165, -2.536]
  Call Extruder 0.01301
  MoveL (T17787) to (121.19, 113.84, 18.9) mm, rotated rx 180 ry 0 rz -180 deg; joints [1.72, 70.375, -36.248, 3.064, -34.165, -2.536]
  Call Extruder 0.13778
  MoveL (T17788) to (117.47, 117.56, 18.9) mm, rotated rx 180 ry 0 rz -180 deg; joints [1.409, 69.45, -34.511, 2.46, -34.964, -2.016]
  Call Extruder 0.00967
  MoveL (T17789) to (117.31, 117.23, 18.9) mm, rotated rx 180 ry 0 rz -180 deg; joints [1.409, 69.45, -34.511, 2.46, -34.964, -2.016]
  Call Extruder 0.14401
  MoveL (T17790) to (121.19, 113.35, 18.9) mm, rotated rx 180 ry 0 rz -180 deg; joints [1.409, 69.45, -34.511, 2.46, -34.964, -2.016]
  Call Extruder 0.01301
  MoveL (T17791) to (121.19, 112.85, 18.9) mm, rotated rx 180 ry 0 rz -180 deg; joints [1.411, 69.278, -34.187, 2.453, -35.116, -2.007]
  Call Extruder 0.15024
  MoveL (T17792) to (117.14, 116.9, 18.9) mm, rotated rx 180 ry 0 rz -180 deg; joints [1.411, 69.278, -34.187, 2.453, -35.116, -2.007]
  Call Extruder 0.00967
  MoveL (T17793) to (116.97, 116.57, 18.9) mm, rotated rx 180 ry 0 rz -180 deg; joints [1.411, 69.278, -34.187, 2.453, -35.116, -2.007]
  Call Extruder 0.15647
  MoveL (T17794) to (121.19, 112.36, 18.9) mm, rotated rx 180 ry 0 rz -180 deg; joints [1.753, 70.288, -36.084, 3.116, -34.243, -2.576]
  Call Extruder 0.01301
  MoveL (T17795) to (121.19, 111.86, 18.9) mm, rotated rx 180 ry 0 rz -180 deg; joints [1.753, 70.288, -36.084, 3.116, -34.243, -2.576]
  Call Extruder 0.1627
  MoveL (T17796) to (116.8, 116.25, 18.9) mm, rotated rx 180 ry 0 rz -180 deg; joints [1.753, 70.288, -36.084, 3.116, -34.243, -2.576]
  Call Extruder 0.00967
  MoveL (T17797) to (116.63, 115.92, 18.9) mm, rotated rx 180 ry 0 rz -180 deg; joints [1.785, 70.201, -35.921, 3.167, -34.32, -2.616]
  Call Extruder 0.16893
  MoveL (T17798) to (121.19, 111.37, 18.9) mm, rotated rx 180 ry 0 rz -180 deg; joints [1.785, 70.201, -35.921, 3.167, -34.32, -2.616]
  Call Extruder 0.01301
  MoveL (T17799) to (121.19, 110.87, 18.9) mm, rotated rx 180 ry 0 rz -180 deg; joints [1.785, 70.201, -35.921, 3.167, -34.32, -2.616]
  Call Extruder 0.17516
  MoveL (T17800) to (116.47, 115.59, 18.9) mm, rotated rx 180 ry 0 rz -180 deg; joints [1.412, 69.106, -33.865, 2.447, -35.266, -1.998]
  Call Extruder 0.00967
  MoveL (T17801) to (116.3, 115.26, 18.9) mm, rotated rx 180 ry 0 rz -180 deg; joints [1.412, 69.106, -33.865, 2.447, -35.266, -1.998]
  Call Extruder 0.18139
  MoveL (T17802) to (121.19, 110.37, 18.9) mm, rotated rx 180 ry 0 rz -180 deg; joints [1.414, 68.936, -33.545, 2.44, -35.416, -1.989]
  Call Extruder 0.01301
  MoveL (T17803) to (121.19, 109.88, 18.9) mm, rotated rx 180 ry 0 rz -180 deg; joints [1.414, 68.936, -33.545, 2.44, -35.416, -1.989]
  Call Extruder 0.18762
  MoveL (T17804) to (116.13, 114.93, 18.9) mm, rotated rx 180 ry 0 rz -180 deg; joints [1.414, 68.936, -33.545, 2.44, -35.416, -1.989]
  Call Extruder 0.00967
  MoveL (T17805) to (115.96, 114.61, 18.9) mm, rotated rx 180 ry 0 rz -180 deg; joints [1.815, 70.109, -35.749, 3.214, -34.402, -2.653]
  Call Extruder 0.19385
  MoveL (T17806) to (121.19, 109.38, 18.9) mm, rotated rx 180 ry 0 rz -180 deg; joints [1.815, 70.109, -35.749, 3.214, -34.402, -2.653]
  Call Extruder 0.01301
  MoveL (T17807) to (121.19, 108.89, 18.9) mm, rotated rx 180 ry 0 rz -180 deg; joints [1.817, 69.932, -35.416, 3.205, -34.558, -2.64]
  Call Extruder 0.20008
  MoveL (T17808) to (115.8, 114.28, 18.9) mm, rotated rx 180 ry 0 rz -180 deg; joints [1.817, 69.932, -35.416, 3.205, -34.558, -2.64]
  Call Extruder 0.00967
  MoveL (T17809) to (115.63, 113.95, 18.9) mm, rotated rx 180 ry 0 rz -180 deg; joints [1.817, 69.932, -35.416, 3.205, -34.558, -2.64]
  Call Extruder 0.20631
  MoveL (T17810) to (121.19, 108.39, 18.9) mm, rotated rx 180 ry 0 rz -180 deg; joints [1.416, 68.767, -33.228, 2.434, -35.564, -1.981]
  Call Extruder 0.01301
  MoveL (T17811) to (121.19, 107.89, 18.9) mm, rotated rx 180 ry 0 rz -180 deg; joints [1.416, 68.767, -33.228, 2.434, -35.564, -1.981]
  Call Extruder 0.21254
  MoveL (T17812) to (115.46, 113.62, 18.9) mm, rotated rx 180 ry 0 rz -180 deg; joints [1.417, 68.6, -32.913, 2.428, -35.711, -1.972]
  Call Extruder 0.00967
  MoveL (T17813) to (115.29, 113.29, 18.9) mm, rotated rx 180 ry 0 rz -180 deg; joints [1.417, 68.6, -32.913, 2.428, -35.711, -1.972]
  Call Extruder 0.21877
  MoveL (T17814) to (121.19, 107.4, 18.9) mm, rotated rx 180 ry 0 rz -180 deg; joints [1.819, 69.756, -35.085, 3.196, -34.712, -2.628]
  Call Extruder 0.01301
  MoveL (T17815) to (121.19, 106.9, 18.9) mm, rotated rx 180 ry 0 rz -180 deg; joints [1.819, 69.756, -35.085, 3.196, -34.712, -2.628]
  Call Extruder 0.225
  MoveL (T17816) to (115.12, 112.97, 18.9) mm, rotated rx 180 ry 0 rz -180 deg; joints [1.819, 69.756, -35.085, 3.196, -34.712, -2.628]
  Call Extruder 0.00967
  MoveL (T17817) to (114.95, 112.64, 18.9) mm, rotated rx 180 ry 0 rz -180 deg; joints [1.821, 69.581, -34.757, 3.187, -34.866, -2.616]
  Call Extruder 0.23123
  MoveL (T17818) to (121.19, 106.41, 18.9) mm, rotated rx 180 ry 0 rz -180 deg; joints [1.821, 69.581, -34.757, 3.187, -34.866, -2.616]
  Call Extruder 0.01301
  MoveL (T17819) to (121.19, 105.91, 18.9) mm, rotated rx 180 ry 0 rz -180 deg; joints [1.419, 68.433, -32.6, 2.422, -35.858, -1.964]
  Call Extruder 0.23746
  MoveL (T17820) to (114.79, 112.31, 18.9) mm, rotated rx 180 ry 0 rz -180 deg; joints [1.419, 68.433, -32.6, 2.422, -35.858, -1.964]
  Call Extruder 0.00967
  MoveL (T17821) to (114.62, 111.98, 18.9) mm, rotated rx 180 ry 0 rz -180 deg; joints [1.419, 68.433, -32.6, 2.422, -35.858, -1.964]
  Call Extruder 0.09826
  MoveL (T17822) to (117.27, 109.33, 18.9) mm, rotated rx 180 ry 0 rz -180 deg; joints [1.42, 68.268, -32.289, 2.417, -36.003, -1.955]
  Call Extruder 0.01301
  MoveL (T17823) to (116.77, 109.33, 18.9) mm, rotated rx 180 ry 0 rz -180 deg; joints [1.42, 68.268, -32.289, 2.417, -36.003, -1.955]
  Call Extruder 0.08609
  MoveL (T17824) to (114.45, 111.65, 18.9) mm, rotated rx 180 ry 0 rz -180 deg; joints [1.42, 68.268, -32.289, 2.417, -36.003, -1.955]
  Call Extruder 0.00967
  MoveL (T17825) to (114.28, 111.33, 18.9) mm, rotated rx 180 ry 0 rz -180 deg; joints [1.823, 69.408, -34.431, 3.179, -35.018, -2.604]
  Call Extruder 0.07391
  MoveL (T17826) to (116.28, 109.33, 18.9) mm, rotated rx 180 ry 0 rz -180 deg; joints [1.823, 69.408, -34.431, 3.179, -35.018, -2.604]
  Call Extruder 0.01301
  MoveL (T17827) to (115.78, 109.33, 18.9) mm, rotated rx 180 ry 0 rz -180 deg; joints [1.825, 69.236, -34.108, 3.17, -35.169, -2.592]
  Call Extruder 0.06174
  MoveL (T17828) to (114.12, 111, 18.9) mm, rotated rx 180 ry 0 rz -180 deg; joints [1.825, 69.236, -34.108, 3.17, -35.169, -2.592]
  Call Extruder 0.00967
  MoveL (T17829) to (113.95, 110.67, 18.9) mm, rotated rx 180 ry 0 rz -180 deg; joints [1.422, 68.103, -31.981, 2.411, -36.147, -1.947]
  Call Extruder 0.04957
  MoveL (T17830) to (115.28, 109.33, 18.9) mm, rotated rx 180 ry 0 rz -180 deg; joints [1.422, 68.103, -31.981, 2.411, -36.147, -1.947]
  Call Extruder 0.01301
  MoveL (T17831) to (114.79, 109.33, 18.9) mm, rotated rx 180 ry 0 rz -180 deg; joints [1.423, 67.94, -31.673, 2.405, -36.291, -1.939]
  Call Extruder 0.03739
  MoveL (T17832) to (113.78, 110.34, 18.9) mm, rotated rx 180 ry 0 rz -180 deg; joints [1.423, 67.94, -31.673, 2.405, -36.291, -1.939]
  Call Extruder 0.00967
  MoveL (T17833) to (113.61, 110.01, 18.9) mm, rotated rx 180 ry 0 rz -180 deg; joints [1.827, 69.065, -33.787, 3.162, -35.319, -2.581]
  Call Extruder 0.02522
  MoveL (T17834) to (114.29, 109.33, 18.9) mm, rotated rx 180 ry 0 rz -180 deg; joints [1.827, 69.065, -33.787, 3.162, -35.319, -2.581]
  Call Extruder 0.01301
  MoveL (T17835) to (113.8, 109.33, 18.9) mm, rotated rx 180 ry 0 rz -180 deg; joints [1.827, 69.065, -33.787, 3.162, -35.319, -2.581]
  Call Extruder 0.01304
  MoveL (T17836) to (113.44, 109.69, 18.9) mm, rotated rx 180 ry 0 rz -180 deg; joints [1.829, 68.895, -33.468, 3.154, -35.468, -2.57]
  Call Extruder 0.00967
  MoveL (T17837) to (113.28, 109.36, 18.9) mm, rotated rx 180 ry 0 rz -180 deg; joints [1.829, 68.895, -33.468, 3.154, -35.468, -2.57]
  Call Extruder 0.00665
  MoveL (T17838) to (113.46, 109.18, 18.9) mm, rotated rx 180 ry 0 rz -180 deg; joints [1.425, 67.778, -31.369, 2.4, -36.433, -1.931]
  Set speed (45.0 mm/s)
  Call Extruder -1.6
  MoveL (T17839) to (113.46, 109.18, 18.9) mm, rotated rx 180 ry 0 rz -180 deg; joints [1.425, 67.778, -31.369, 2.4, -36.433, -1.931]
  Set speed (120.0 mm/s)
  MoveL (T17840) to (113.46, 109.18, 18.9) mm, rotated rx 180 ry 0 rz -180 deg; joints [1.427, 67.616, -31.065, 2.395, -36.575, -1.923]
  Call Extruder -0.09026
  MoveL (T17841) to (113.28, 109.36, 18.9) mm, rotated rx 180 ry 0 rz -180 deg; joints [1.427, 67.616, -31.065, 2.395, -36.575, -1.923]
  Call Extruder -0.13128
  MoveL (T17842) to (113.44, 109.69, 18.9) mm, rotated rx 180 ry 0 rz -180 deg; joints [1.427, 67.616, -31.065, 2.395, -36.575, -1.923]
  Call Extruder -0.15846
  MoveL (T17843) to (113.76, 109.37, 18.9) mm, rotated rx 180 ry 0 rz -180 deg; joints [1.69, 68.331, -32.408, 2.879, -35.958, -2.331]
  Set speed (45.0 mm/s)
  Call Extruder -0.02
  MoveL (T17844) to (113.76, 109.37, 18.9) mm, rotated rx 180 ry 0 rz -180 deg; joints [1.69, 68.331, -32.408, 2.879, -35.958, -2.331]
  Set speed (150.0 mm/s)
  MoveL (T17845) to (113.76, 109.37, 20.9) mm, rotated rx 180 ry 0 rz -180 deg; joints [1.723, 68.251, -32.257, 2.93, -36.029, -2.37]
  MoveL (T17846) to (117.77, 108.83, 20.9) mm, rotated rx 180 ry 0 rz -180 deg; joints [1.723, 68.251, -32.257, 2.93, -36.029, -2.37]
  MoveL (T17847) to (117.77, 108.83, 18.9) mm, rotated rx 180 ry 0 rz -180 deg; joints [1.723, 68.251, -32.257, 2.93, -36.029, -2.37]
  Set speed (40.0 mm/s)
  Call Extruder 2.0
  MoveL (T17848) to (117.77, 108.83, 18.9) mm, rotated rx 180 ry 0 rz -180 deg; joints [1.428, 67.456, -30.765, 2.389, -36.715, -1.916]
  Set speed (25.0 mm/s)
  MoveL (T17849) to (117.77, 108.83, 18.9) mm, rotated rx 180 ry 0 rz -180 deg; joints [1.43, 67.297, -30.465, 2.384, -36.855, -1.908]
  Call Extruder 0.12676
  MoveL (T17850) to (121.19, 105.42, 18.9) mm, rotated rx 180 ry 0 rz -180 deg; joints [1.43, 67.297, -30.465, 2.384, -36.855, -1.908]
  Call Extruder 0.01301
  MoveL (T17851) to (121.19, 104.92, 18.9) mm, rotated rx 180 ry 0 rz -180 deg; joints [1.755, 68.171, -32.107, 2.98, -36.101, -2.409]
  Call Extruder 0.12098
  MoveL (T17852) to (117.93, 108.18, 18.9) mm, rotated rx 180 ry 0 rz -180 deg; joints [1.755, 68.171, -32.107, 2.98, -36.101, -2.409]
  Call Extruder 0.01301
  MoveL (T17853) to (117.93, 107.68, 18.9) mm, rotated rx 180 ry 0 rz -180 deg; joints [1.755, 68.171, -32.107, 2.98, -36.101, -2.409]
  Call Extruder 0.12098
  MoveL (T17854) to (121.19, 104.42, 18.9) mm, rotated rx 180 ry 0 rz -180 deg; joints [1.788, 68.091, -31.958, 3.031, -36.172, -2.447]
  Call Extruder 0.01301
  MoveL (T17855) to (121.19, 103.93, 18.9) mm, rotated rx 180 ry 0 rz -180 deg; joints [1.788, 68.091, -31.958, 3.031, -36.172, -2.447]
  Call Extruder 0.12098
  MoveL (T17856) to (117.93, 107.19, 18.9) mm, rotated rx 180 ry 0 rz -180 deg; joints [1.431, 67.138, -30.168, 2.379, -36.994, -1.901]
  Call Extruder 0.01301
  MoveL (T17857) to (117.93, 106.69, 18.9) mm, rotated rx 180 ry 0 rz -180 deg; joints [1.431, 67.138, -30.168, 2.379, -36.994, -1.901]
  Call Extruder 0.10678
  MoveL (T17858) to (120.8, 103.81, 18.9) mm, rotated rx 180 ry 0 rz -180 deg; joints [1.431, 67.138, -30.168, 2.379, -36.994, -1.901]
  Call Extruder 0.01301
  MoveL (T17859) to (120.31, 103.81, 18.9) mm, rotated rx 180 ry 0 rz -180 deg; joints [1.433, 66.981, -29.872, 2.374, -37.132, -1.893]
  Call Extruder 0.08838
  MoveL (T17860) to (117.93, 106.19, 18.9) mm, rotated rx 180 ry 0 rz -180 deg; joints [1.433, 66.981, -29.872, 2.374, -37.132, -1.893]
  Call Extruder 0.01301
  MoveL (T17861) to (117.93, 105.7, 18.9) mm, rotated rx 180 ry 0 rz -180 deg; joints [1.821, 68.012, -31.809, 3.081, -36.242, -2.486]
  Call Extruder 0.06998
  MoveL (T17862) to (119.81, 103.81, 18.9) mm, rotated rx 180 ry 0 rz -180 deg; joints [1.821, 68.012, -31.809, 3.081, -36.242, -2.486]
  Call Extruder 0.01301
  MoveL (T17863) to (119.32, 103.81, 18.9) mm, rotated rx 180 ry 0 rz -180 deg; joints [1.821, 68.012, -31.809, 3.081, -36.242, -2.486]
  Call Extruder 0.05157
  MoveL (T17864) to (117.93, 105.2, 18.9) mm, rotated rx 180 ry 0 rz -180 deg; joints [1.838, 67.97, -31.729, 3.108, -36.281, -2.506]
  Call Extruder 0.01301
  MoveL (T17865) to (117.93, 104.71, 18.9) mm, rotated rx 180 ry 0 rz -180 deg; joints [1.838, 67.97, -31.729, 3.108, -36.281, -2.506]
  Call Extruder 0.03317
  MoveL (T17866) to (118.82, 103.81, 18.9) mm, rotated rx 180 ry 0 rz -180 deg; joints [1.838, 67.97, -31.729, 3.108, -36.281, -2.506]
  Call Extruder 0.01301
  MoveL (T17867) to (118.32, 103.81, 18.9) mm, rotated rx 180 ry 0 rz -180 deg; joints [1.838, 67.97, -31.729, 3.108, -36.281, -2.506]
  Call Extruder 0.02054
  MoveL (T17868) to (117.77, 104.37, 18.9) mm, rotated rx 180 ry 0 rz -180 deg; joints [1.838, 67.97, -31.729, 3.108, -36.281, -2.506]
  Set speed (45.0 mm/s)
  Call Extruder -1.6
  MoveL (T17869) to (117.77, 104.37, 18.9) mm, rotated rx 180 ry 0 rz -180 deg; joints [1.842, 67.9, -31.599, 3.109, -36.341, -2.505]
  Set speed (120.0 mm/s)
  MoveL (T17870) to (117.77, 104.37, 18.9) mm, rotated rx 180 ry 0 rz -180 deg; joints [1.842, 67.9, -31.599, 3.109, -36.341, -2.505]
  Call Extruder -0.27887
  MoveL (T17871) to (118.32, 103.81, 18.9) mm, rotated rx 180 ry 0 rz -180 deg; joints [1.435, 66.824, -29.578, 2.369, -37.27, -1.886]
  Call Extruder -0.10113
  MoveL (T17872) to (118.61, 103.81, 18.9) mm, rotated rx 180 ry 0 rz -180 deg; joints [1.435, 66.824, -29.578, 2.369, -37.27, -1.886]
  Set speed (45.0 mm/s)
  Call Extruder -0.02
  MoveL (T17873) to (118.61, 103.81, 18.9) mm, rotated rx 180 ry 0 rz -180 deg; joints [1.435, 66.824, -29.578, 2.369, -37.27, -1.886]
  Set speed (150.0 mm/s)
  MoveL (T17874) to (118.61, 103.81, 20.9) mm, rotated rx 180 ry 0 rz -180 deg; joints [1.436, 66.669, -29.286, 2.365, -37.406, -1.879]
  MoveL (T17875) to (109.4, 105.47, 20.9) mm, rotated rx 180 ry 0 rz -180 deg; joints [1.436, 66.669, -29.286, 2.365, -37.406, -1.879]
  MoveL (T17876) to (109.4, 105.47, 19.1) mm, rotated rx 180 ry 0 rz -180 deg; joints [1.844, 67.739, -31.295, 3.102, -36.483, -2.495]
  Set speed (40.0 mm/s)
  Call Extruder 2.0
  MoveL (T17877) to (109.4, 105.47, 19.1) mm, rotated rx 180 ry 0 rz -180 deg; joints [1.844, 67.739, -31.295, 3.102, -36.483, -2.495]
  Call Extruder 0.25145
  MoveL (T17878) to (117.65, 105.47, 19.1) mm, rotated rx 180 ry 0 rz -180 deg; joints [1.844, 67.739, -31.295, 3.102, -36.483, -2.495]
  Call Extruder 0.10939
  MoveL (T17879) to (117.65, 109.06, 19.1) mm, rotated rx 180 ry 0 rz -180 deg; joints [1.846, 67.577, -30.992, 3.095, -36.625, -2.485]
  Call Extruder 0.14732
  MoveL (T17880) to (112.81, 109.06, 19.1) mm, rotated rx 180 ry 0 rz -180 deg; joints [1.438, 66.514, -28.995, 2.36, -37.542, -1.872]
  Call Extruder 0.31102
  MoveL (T17881) to (117.47, 118.15, 19.1) mm, rotated rx 180 ry 0 rz -180 deg; joints [1.438, 66.514, -28.995, 2.36, -37.542, -1.872]
  Call Extruder 0.05209
  MoveL (T17882) to (117.47, 119.86, 19.1) mm, rotated rx 180 ry 0 rz -180 deg; joints [1.438, 66.514, -28.995, 2.36, -37.542, -1.872]
  Call Extruder 0.29244
  MoveL (T17883) to (107.87, 119.86, 19.1) mm, rotated rx 180 ry 0 rz -180 deg; joints [1.438, 66.514, -28.995, 2.36, -37.542, -1.872]
  Call Extruder 0.10939
  MoveL (T17884) to (107.87, 116.27, 19.1) mm, rotated rx 180 ry 0 rz -180 deg; joints [1.439, 66.36, -28.707, 2.355, -37.677, -1.865]
  Call Extruder 0.13869
  MoveL (T17885) to (112.42, 116.27, 19.1) mm, rotated rx 180 ry 0 rz -180 deg; joints [1.439, 66.36, -28.707, 2.355, -37.677, -1.865]
  Call Extruder 0.31084
  MoveL (T17886) to (107.78, 107.18, 19.1) mm, rotated rx 180 ry 0 rz -180 deg; joints [1.439, 66.36, -28.707, 2.355, -37.677, -1.865]
  Call Extruder 0.05206
  MoveL (T17887) to (107.78, 105.47, 19.1) mm, rotated rx 180 ry 0 rz -180 deg; joints [1.848, 67.417, -30.692, 3.088, -36.765, -2.475]
  Call Extruder 0.04735
  MoveL (T17888) to (109.34, 105.47, 19.1) mm, rotated rx 180 ry 0 rz -180 deg; joints [1.848, 67.417, -30.692, 3.088, -36.765, -2.475]
  Set speed (150.0 mm/s)
  MoveL (T17889) to (109, 105.88, 19.1) mm, rotated rx 180 ry 0 rz -180 deg; joints [1.85, 67.258, -30.394, 3.082, -36.905, -2.465]
  Set speed (40.0 mm/s)
  MoveL (T17890) to (109, 105.88, 19.1) mm, rotated rx 180 ry 0 rz -180 deg; joints [1.85, 67.258, -30.394, 3.082, -36.905, -2.465]
  Call Extruder 0.25124
  MoveL (T17891) to (117.24, 105.88, 19.1) mm, rotated rx 180 ry 0 rz -180 deg; joints [1.456, 66.246, -28.492, 2.378, -37.778, -1.88]
  Call Extruder 0.08459
  MoveL (T17892) to (117.24, 108.65, 19.1) mm, rotated rx 180 ry 0 rz -180 deg; joints [1.456, 66.246, -28.492, 2.378, -37.778, -1.88]
  Call Extruder 0.1552
  MoveL (T17893) to (112.15, 108.65, 19.1) mm, rotated rx 180 ry 0 rz -180 deg; joints [1.521, 66.25, -28.499, 2.483, -37.776, -1.963]
  Call Extruder 0.32831
  MoveL (T17894) to (117.06, 118.25, 19.1) mm, rotated rx 180 ry 0 rz -180 deg; joints [1.521, 66.25, -28.499, 2.483, -37.776, -1.963]
  Call Extruder 0.0367
  MoveL (T17895) to (117.06, 119.45, 19.1) mm, rotated rx 180 ry 0 rz -180 deg; joints [1.521, 66.25, -28.499, 2.483, -37.776, -1.963]
  Call Extruder 0.26763
  MoveL (T17896) to (108.27, 119.45, 19.1) mm, rotated rx 180 ry 0 rz -180 deg; joints [1.852, 67.1, -30.096, 3.075, -37.044, -2.455]
  Call Extruder 0.08459
  MoveL (T17897) to (108.27, 116.67, 19.1) mm, rotated rx 180 ry 0 rz -180 deg; joints [1.852, 67.1, -30.096, 3.075, -37.044, -2.455]
  Call Extruder 0.14654
  MoveL (T17898) to (113.08, 116.67, 19.1) mm, rotated rx 180 ry 0 rz -180 deg; joints [1.854, 66.943, -29.801, 3.069, -37.181, -2.446]
  Call Extruder 0.32811
  MoveL (T17899) to (108.19, 107.08, 19.1) mm, rotated rx 180 ry 0 rz -180 deg; joints [1.854, 66.943, -29.801, 3.069, -37.181, -2.446]
  Call Extruder 0.03668
  MoveL (T17900) to (108.19, 105.88, 19.1) mm, rotated rx 180 ry 0 rz -180 deg; joints [1.585, 66.254, -28.508, 2.588, -37.775, -2.046]
  Call Extruder 0.02276
  MoveL (T17901) to (108.94, 105.88, 19.1) mm, rotated rx 180 ry 0 rz -180 deg; joints [1.585, 66.254, -28.508, 2.588, -37.775, -2.046]
  Set speed (150.0 mm/s)
  MoveL (T17902) to (108.6, 106.28, 19.1) mm, rotated rx 180 ry 0 rz -180 deg; joints [1.585, 66.254, -28.508, 2.588, -37.775, -2.046]
  Set speed (25.0 mm/s)
  MoveL (T17903) to (108.6, 106.28, 19.1) mm, rotated rx 180 ry 0 rz -180 deg; joints [1.647, 66.258, -28.515, 2.69, -37.773, -2.127]
  Call Extruder 0.25102
  MoveL (T17904) to (116.84, 106.28, 19.1) mm, rotated rx 180 ry 0 rz -180 deg; joints [1.647, 66.258, -28.515, 2.69, -37.773, -2.127]
  Call Extruder 0.05979
  MoveL (T17905) to (116.84, 108.25, 19.1) mm, rotated rx 180 ry 0 rz -180 deg; joints [1.651, 66.262, -28.523, 2.696, -37.77, -2.132]
  Call Extruder 0.16307
  MoveL (T17906) to (111.48, 108.25, 19.1) mm, rotated rx 180 ry 0 rz -180 deg; joints [1.651, 66.262, -28.523, 2.696, -37.77, -2.132]
  Call Extruder 0.3456
  MoveL (T17907) to (116.65, 118.34, 19.1) mm, rotated rx 180 ry 0 rz -180 deg; joints [1.651, 66.262, -28.523, 2.696, -37.77, -2.132]
  Call Extruder 0.02131
  MoveL (T17908) to (116.65, 119.04, 19.1) mm, rotated rx 180 ry 0 rz -180 deg; joints [1.875, 66.836, -29.601, 3.097, -37.276, -2.465]
  Call Extruder 0.24283
  MoveL (T17909) to (108.68, 119.04, 19.1) mm, rotated rx 180 ry 0 rz -180 deg; joints [1.875, 66.836, -29.601, 3.097, -37.276, -2.465]
  Call Extruder 0.05979
  MoveL (T17910) to (108.68, 117.08, 19.1) mm, rotated rx 180 ry 0 rz -180 deg; joints [1.875, 66.836, -29.601, 3.097, -37.276, -2.465]
  Call Extruder 0.15438
  MoveL (T17911) to (113.75, 117.08, 19.1) mm, rotated rx 180 ry 0 rz -180 deg; joints [1.875, 66.836, -29.601, 3.097, -37.276, -2.465]
  Call Extruder 0.34538
  MoveL (T17912) to (108.6, 106.98, 19.1) mm, rotated rx 180 ry 0 rz -180 deg; joints [1.875, 66.836, -29.601, 3.097, -37.276, -2.465]
  Call Extruder 0.01947
  MoveL (T17913) to (108.6, 106.34, 19.1) mm, rotated rx 180 ry 0 rz -180 deg; joints [1.875, 66.836, -29.601, 3.097, -37.276, -2.465]
  Set speed (150.0 mm/s)
  MoveL (T17914) to (108.54, 105.89, 19.1) mm, rotated rx 180 ry 0 rz -180 deg; joints [1.875, 66.836, -29.601, 3.097, -37.276, -2.465]
  Set speed (45.0 mm/s)
  Call Extruder -1.6
  MoveL (T17915) to (108.54, 105.89, 19.1) mm, rotated rx 180 ry 0 rz -180 deg; joints [1.875, 66.836, -29.601, 3.097, -37.276, -2.465]
  Set speed (120.0 mm/s)
  MoveL (T17916) to (108.54, 105.89, 19.1) mm, rotated rx 180 ry 0 rz -180 deg; joints [1.875, 66.836, -29.601, 3.097, -37.276, -2.465]
  Call Extruder -0.38
  MoveL (T17917) to (109.66, 106.33, 19.1) mm, rotated rx 180 ry 0 rz -180 deg; joints [1.796, 66.632, -29.218, 2.955, -37.451, -2.347]
  Set speed (45.0 mm/s)
  Call Extruder -0.02
  MoveL (T17918) to (109.66, 106.33, 19.1) mm, rotated rx 180 ry 0 rz -180 deg; joints [1.796, 66.632, -29.218, 2.955, -37.451, -2.347]
  Set speed (150.0 mm/s)
  MoveL (T17919) to (109.66, 106.33, 21.1) mm, rotated rx 180 ry 0 rz -180 deg; joints [1.796, 66.632, -29.218, 2.955, -37.451, -2.347]
  MoveL (T17920) to (104.34, 103.54, 21.1) mm, rotated rx 180 ry 0 rz -180 deg; joints [1.796, 66.632, -29.218, 2.955, -37.451, -2.347]
  MoveL (T17921) to (104.34, 103.54, 19.1) mm, rotated rx 180 ry 0 rz -180 deg; joints [1.796, 66.632, -29.218, 2.955, -37.451, -2.347]
  Set speed (40.0 mm/s)
  Call Extruder 2.0
  MoveL (T17922) to (104.34, 103.54, 19.1) mm, rotated rx 180 ry 0 rz -180 deg; joints [1.796, 66.632, -29.218, 2.955, -37.451, -2.347]
  Call Extruder 0.52159
  MoveL (T17923) to (121.46, 103.54, 19.1) mm, rotated rx 180 ry 0 rz -180 deg; joints [3.301, 66.726, -29.799, 5.484, -37.054, -4.381]
  Call Extruder 0.54596
  MoveL (T17924) to (121.46, 121.46, 19.1) mm, rotated rx 180 ry 0 rz -180 deg; joints [3.301, 66.962, -29.836, 5.459, -37.251, -4.35]
  Call Extruder 0.54596
  MoveL (T17925) to (103.54, 121.46, 19.1) mm, rotated rx 180 ry 0 rz -180 deg; joints [3.301, 66.962, -29.836, 5.459, -37.251, -4.35]
  Call Extruder 0.54596
  MoveL (T17926) to (103.54, 103.54, 19.1) mm, rotated rx 180 ry 0 rz -180 deg; joints [3.301, 66.962, -29.836, 5.459, -37.251, -4.35]
  Call Extruder 0.02254
  MoveL (T17927) to (104.28, 103.54, 19.1) mm, rotated rx 180 ry 0 rz -180 deg; joints [3.301, 66.962, -29.836, 5.459, -37.251, -4.35]
  Set speed (150.0 mm/s)
  MoveL (T17928) to (103.53, 103.13, 19.1) mm, rotated rx 180 ry 0 rz -180 deg; joints [3.301, 66.962, -29.836, 5.459, -37.251, -4.35]
  Set speed (40.0 mm/s)
  MoveL (T17929) to (103.53, 103.13, 19.1) mm, rotated rx 180 ry 0 rz -180 deg; joints [3.301, 66.962, -29.836, 5.459, -37.251, -4.35]
  Call Extruder 0.55858
  MoveL (T17930) to (121.87, 103.13, 19.1) mm, rotated rx 180 ry 0 rz -180 deg; joints [3.301, 66.962, -29.836, 5.459, -37.251, -4.35]
  Call Extruder 0.57077
  MoveL (T17931) to (121.87, 121.87, 19.1) mm, rotated rx 180 ry 0 rz -180 deg; joints [3.301, 66.962, -29.836, 5.459, -37.251, -4.35]
  Call Extruder 0.57077
  MoveL (T17932) to (103.13, 121.87, 19.1) mm, rotated rx 180 ry 0 rz -180 deg; joints [3.301, 66.962, -29.836, 5.459, -37.251, -4.35]
  Call Extruder 0.57077
  MoveL (T17933) to (103.13, 103.13, 19.1) mm, rotated rx 180 ry 0 rz -180 deg; joints [3.301, 66.962, -29.836, 5.459, -37.251, -4.35]
  Call Extruder 0.01036
  MoveL (T17934) to (103.47, 103.13, 19.1) mm, rotated rx 180 ry 0 rz -180 deg; joints [3.316, 66.324, -28.639, 5.415, -37.809, -4.283]
  Set speed (150.0 mm/s)
  MoveL (T17935) to (102.72, 102.81, 19.1) mm, rotated rx 180 ry 0 rz -180 deg; joints [3.316, 66.324, -28.639, 5.415, -37.809, -4.283]
  Set speed (25.0 mm/s)
  MoveL (T17936) to (102.72, 102.81, 19.1) mm, rotated rx 180 ry 0 rz -180 deg; joints [1.863, 69.742, -35.059, 3.271, -34.727, -2.689]
  Call Extruder 0.00259
  MoveL (T17937) to (102.72, 102.72, 19.1) mm, rotated rx 180 ry 0 rz -180 deg; joints [1.863, 69.742, -35.059, 3.271, -34.727, -2.689]
  Call Extruder 0.59557
  MoveL (T17938) to (122.28, 102.72, 19.1) mm, rotated rx 180 ry 0 rz -180 deg; joints [1.863, 69.742, -35.059, 3.271, -34.727, -2.689]
  Call Extruder 0.59557
  MoveL (T17939) to (122.28, 122.28, 19.1) mm, rotated rx 180 ry 0 rz -180 deg; joints [1.863, 69.742, -35.059, 3.271, -34.727, -2.689]
  Call Extruder 0.59557
  MoveL (T17940) to (102.72, 122.28, 19.1) mm, rotated rx 180 ry 0 rz -180 deg; joints [1.861, 69.894, -35.345, 3.279, -34.593, -2.7]
  Call Extruder 0.59115
  MoveL (T17941) to (102.72, 102.87, 19.1) mm, rotated rx 180 ry 0 rz -180 deg; joints [1.915, 70.056, -35.65, 3.386, -34.453, -2.793]
  Set speed (150.0 mm/s)
  MoveL (T17942) to (102.78, 102.75, 19.1) mm, rotated rx 180 ry 0 rz -180 deg; joints [1.915, 70.056, -35.65, 3.386, -34.453, -2.793]
  Set speed (45.0 mm/s)
  Call Extruder -1.6
  MoveL (T17943) to (102.78, 102.75, 19.1) mm, rotated rx 180 ry 0 rz -180 deg; joints [1.915, 70.056, -35.65, 3.386, -34.453, -2.793]
  Set speed (120.0 mm/s)
  MoveL (T17944) to (102.78, 102.75, 19.1) mm, rotated rx 180 ry 0 rz -180 deg; joints [1.915, 70.056, -35.65, 3.386, -34.453, -2.793]
  Call Extruder -0.05166
  MoveL (T17945) to (102.72, 102.72, 19.1) mm, rotated rx 180 ry 0 rz -180 deg; joints [1.803, 70.356, -36.212, 3.21, -34.185, -2.656]
  Call Extruder -0.32834
  MoveL (T17946) to (103.65, 102.72, 19.1) mm, rotated rx 180 ry 0 rz -180 deg; joints [1.803, 70.356, -36.212, 3.21, -34.185, -2.656]
  Set speed (45.0 mm/s)
  Call Extruder -0.02
  MoveL (T17947) to (103.65, 102.72, 19.1) mm, rotated rx 180 ry 0 rz -180 deg; joints [1.794, 70.416, -36.326, 3.198, -34.132, -2.648]
  Set speed (150.0 mm/s)
  MoveL (T17948) to (103.65, 102.72, 21.1) mm, rotated rx 180 ry 0 rz -180 deg; joints [1.794, 70.416, -36.326, 3.198, -34.132, -2.648]
  MoveL (T17949) to (120.51, 103.66, 21.1) mm, rotated rx 180 ry 0 rz -180 deg; joints [1.787, 71.045, -37.507, 3.232, -33.58, -2.693]
  MoveL (T17950) to (120.51, 103.66, 19.1) mm, rotated rx 180 ry 0 rz -180 deg; joints [1.787, 71.045, -37.507, 3.232, -33.58, -2.693]
  Set speed (40.0 mm/s)
  Call Extruder 2.0
  MoveL (T17951) to (120.51, 103.66, 19.1) mm, rotated rx 180 ry 0 rz -180 deg; joints [1.787, 71.045, -37.507, 3.232, -33.58, -2.693]
  Call Extruder 0.02815
  MoveL (T17952) to (121.16, 104.31, 19.1) mm, rotated rx 180 ry 0 rz -180 deg; joints [1.763, 71.043, -37.503, 3.188, -33.581, -2.657]
  Call Extruder 0.01786
  MoveL (T17953) to (121.16, 104.89, 19.1) mm, rotated rx 180 ry 0 rz -180 deg; joints [1.763, 71.043, -37.503, 3.188, -33.581, -2.657]
  Call Extruder 0.04544
  MoveL (T17954) to (120.11, 103.84, 19.1) mm, rotated rx 180 ry 0 rz -180 deg; joints [1.763, 71.043, -37.503, 3.188, -33.581, -2.657]
  Call Extruder 0.01786
  MoveL (T17955) to (119.53, 103.84, 19.1) mm, rotated rx 180 ry 0 rz -180 deg; joints [1.659, 70.715, -36.888, 2.977, -33.863, -2.473]
  Call Extruder 0.0707
  MoveL (T17956) to (121.16, 105.47, 19.1) mm, rotated rx 180 ry 0 rz -180 deg; joints [1.659, 70.715, -36.888, 2.977, -33.863, -2.473]
  Call Extruder 0.01786
  MoveL (T17957) to (121.16, 106.05, 19.1) mm, rotated rx 180 ry 0 rz -180 deg; joints [1.659, 70.715, -36.888, 2.977, -33.863, -2.473]
  Call Extruder 0.09595
  MoveL (T17958) to (118.95, 103.84, 19.1) mm, rotated rx 180 ry 0 rz -180 deg; joints [1.659, 70.715, -36.888, 2.977, -33.863, -2.473]
  Call Extruder 0.01786
  MoveL (T17959) to (118.37, 103.84, 19.1) mm, rotated rx 180 ry 0 rz -180 deg; joints [1.628, 70.8, -37.048, 2.928, -33.787, -2.434]
  Call Extruder 0.12121
  MoveL (T17960) to (121.16, 106.63, 19.1) mm, rotated rx 180 ry 0 rz -180 deg; joints [1.628, 70.8, -37.048, 2.928, -33.787, -2.434]
  Call Extruder 0.01786
  MoveL (T17961) to (121.16, 107.21, 19.1) mm, rotated rx 180 ry 0 rz -180 deg; joints [1.607, 70.824, -37.093, 2.892, -33.765, -2.404]
  Call Extruder 0.14646
  MoveL (T17962) to (117.79, 103.84, 19.1) mm, rotated rx 180 ry 0 rz -180 deg; joints [1.607, 70.824, -37.093, 2.892, -33.765, -2.404]
  Call Extruder 0.01786
  MoveL (T17963) to (117.21, 103.84, 19.1) mm, rotated rx 180 ry 0 rz -180 deg; joints [1.607, 70.824, -37.093, 2.892, -33.765, -2.404]
  Call Extruder 0.17172
  MoveL (T17964) to (121.16, 107.79, 19.1) mm, rotated rx 180 ry 0 rz -180 deg; joints [1.467, 70.814, -37.073, 2.639, -33.769, -2.194]
  Call Extruder 0.01786
  MoveL (T17965) to (121.16, 108.38, 19.1) mm, rotated rx 180 ry 0 rz -180 deg; joints [1.467, 70.814, -37.073, 2.639, -33.769, -2.194]
  Call Extruder 0.19697
  MoveL (T17966) to (116.62, 103.84, 19.1) mm, rotated rx 180 ry 0 rz -180 deg; joints [1.467, 70.814, -37.073, 2.639, -33.769, -2.194]
  Call Extruder 0.01786
  MoveL (T17967) to (116.04, 103.84, 19.1) mm, rotated rx 180 ry 0 rz -180 deg; joints [1.396, 71.012, -37.446, 2.524, -33.592, -2.103]
  Call Extruder 0.0573
  MoveL (T17968) to (117.36, 105.16, 19.1) mm, rotated rx 180 ry 0 rz -180 deg; joints [1.396, 71.012, -37.446, 2.524, -33.592, -2.103]
  Call Extruder 0.01786
  MoveL (T17969) to (116.78, 105.16, 19.1) mm, rotated rx 180 ry 0 rz -180 deg; joints [1.396, 71.012, -37.446, 2.524, -33.592, -2.103]
  Call Extruder 0.0573
  MoveL (T17970) to (115.46, 103.84, 19.1) mm, rotated rx 180 ry 0 rz -180 deg; joints [1.652, 71.033, -37.484, 2.988, -33.584, -2.49]
  Call Extruder 0.01786
  MoveL (T17971) to (114.88, 103.84, 19.1) mm, rotated rx 180 ry 0 rz -180 deg; joints [1.652, 71.033, -37.484, 2.988, -33.584, -2.49]
  Call Extruder 0.0573
  MoveL (T17972) to (116.2, 105.16, 19.1) mm, rotated rx 180 ry 0 rz -180 deg; joints [1.652, 71.033, -37.484, 2.988, -33.584, -2.49]
  Call Extruder 0.01786
  MoveL (T17973) to (115.62, 105.16, 19.1) mm, rotated rx 180 ry 0 rz -180 deg; joints [1.652, 71.033, -37.484, 2.988, -33.584, -2.49]
  Call Extruder 0.0573
  MoveL (T17974) to (114.3, 103.84, 19.1) mm, rotated rx 180 ry 0 rz -180 deg; joints [1.652, 71.033, -37.484, 2.988, -33.584, -2.49]
  Call Extruder 0.01786
  MoveL (T17975) to (113.72, 103.84, 19.1) mm, rotated rx 180 ry 0 rz -180 deg; joints [1.652, 71.033, -37.484, 2.988, -33.584, -2.49]
  Call Extruder 0.0573
  MoveL (T17976) to (115.04, 105.16, 19.1) mm, rotated rx 180 ry 0 rz -180 deg; joints [1.652, 71.033, -37.484, 2.988, -33.584, -2.49]
  Call Extruder 0.01786
  MoveL (T17977) to (114.46, 105.16, 19.1) mm, rotated rx 180 ry 0 rz -180 deg; joints [1.54, 71.023, -37.467, 2.785, -33.588, -2.321]
  Call Extruder 0.0573
  MoveL (T17978) to (113.14, 103.84, 19.1) mm, rotated rx 180 ry 0 rz -180 deg; joints [1.54, 71.023, -37.467, 2.785, -33.588, -2.321]
  Call Extruder 0.01786
  MoveL (T17979) to (112.56, 103.84, 19.1) mm, rotated rx 180 ry 0 rz -180 deg; joints [1.54, 71.023, -37.467, 2.785, -33.588, -2.321]
  Call Extruder 0.0573
  MoveL (T17980) to (113.88, 105.16, 19.1) mm, rotated rx 180 ry 0 rz -180 deg; joints [1.54, 71.023, -37.467, 2.785, -33.588, -2.321]
  Call Extruder 0.01786
  MoveL (T17981) to (113.3, 105.16, 19.1) mm, rotated rx 180 ry 0 rz -180 deg; joints [1.54, 71.023, -37.467, 2.785, -33.588, -2.321]
  Call Extruder 0.0573
  MoveL (T17982) to (111.98, 103.84, 19.1) mm, rotated rx 180 ry 0 rz -180 deg; joints [1.54, 71.023, -37.467, 2.785, -33.588, -2.321]
  Call Extruder 0.01786
  MoveL (T17983) to (111.4, 103.84, 19.1) mm, rotated rx 180 ry 0 rz -180 deg; joints [1.54, 71.023, -37.467, 2.785, -33.588, -2.321]
  Call Extruder 0.0573
  MoveL (T17984) to (112.72, 105.16, 19.1) mm, rotated rx 180 ry 0 rz -180 deg; joints [1.54, 71.023, -37.467, 2.785, -33.588, -2.321]
  Call Extruder 0.01786
  MoveL (T17985) to (112.13, 105.16, 19.1) mm, rotated rx 180 ry 0 rz -180 deg; joints [1.54, 70.791, -37.424, 2.799, -33.398, -2.338]
  Call Extruder 0.0573
  MoveL (T17986) to (110.81, 103.84, 19.1) mm, rotated rx 180 ry 0 rz -180 deg; joints [1.407, 66.028, -28.491, 2.309, -37.56, -1.831]
  Call Extruder 0.01786
  MoveL (T17987) to (110.23, 103.84, 19.1) mm, rotated rx 180 ry 0 rz -180 deg; joints [1.407, 66.241, -28.523, 2.3, -37.74, -1.819]
  Call Extruder 0.0573
  MoveL (T17988) to (111.55, 105.16, 19.1) mm, rotated rx 180 ry 0 rz -180 deg; joints [1.407, 66.241, -28.523, 2.3, -37.74, -1.819]
  Call Extruder 0.01786
  MoveL (T17989) to (110.97, 105.16, 19.1) mm, rotated rx 180 ry 0 rz -180 deg; joints [1.407, 66.241, -28.523, 2.3, -37.74, -1.819]
  Call Extruder 0.0573
  MoveL (T17990) to (109.65, 103.84, 19.1) mm, rotated rx 180 ry 0 rz -180 deg; joints [1.407, 66.241, -28.523, 2.3, -37.74, -1.819]
  Call Extruder 0.01786
  MoveL (T17991) to (109.07, 103.84, 19.1) mm, rotated rx 180 ry 0 rz -180 deg; joints [1.407, 66.241, -28.523, 2.3, -37.74, -1.819]
  Call Extruder 0.0573
  MoveL (T17992) to (110.39, 105.16, 19.1) mm, rotated rx 180 ry 0 rz -180 deg; joints [1.407, 66.241, -28.523, 2.3, -37.74, -1.819]
  Call Extruder 0.01786
  MoveL (T17993) to (109.81, 105.16, 19.1) mm, rotated rx 180 ry 0 rz -180 deg; joints [1.407, 66.241, -28.523, 2.3, -37.74, -1.819]
  Call Extruder 0.0573
  MoveL (T17994) to (108.49, 103.84, 19.1) mm, rotated rx 180 ry 0 rz -180 deg; joints [1.407, 66.241, -28.523, 2.3, -37.74, -1.819]
  Call Extruder 0.01786
  MoveL (T17995) to (107.91, 103.84, 19.1) mm, rotated rx 180 ry 0 rz -180 deg; joints [1.407, 66.241, -28.523, 2.3, -37.74, -1.819]
  Call Extruder 0.0573
  MoveL (T17996) to (109.23, 105.16, 19.1) mm, rotated rx 180 ry 0 rz -180 deg; joints [1.407, 66.241, -28.523, 2.3, -37.74, -1.819]
  Call Extruder 0.01786
  MoveL (T17997) to (108.65, 105.16, 19.1) mm, rotated rx 180 ry 0 rz -180 deg; joints [1.407, 66.241, -28.523, 2.3, -37.74, -1.819]
  Call Extruder 0.0573
  MoveL (T17998) to (107.33, 103.84, 19.1) mm, rotated rx 180 ry 0 rz -180 deg; joints [1.407, 66.241, -28.523, 2.3, -37.74, -1.819]
  Call Extruder 0.01786
  MoveL (T17999) to (106.75, 103.84, 19.1) mm, rotated rx 180 ry 0 rz -180 deg; joints [1.363, 71.082, -37.617, 2.471, -33.49, -2.061]
  Call Extruder 0.0573
  MoveL (T18000) to (108.07, 105.16, 19.1) mm, rotated rx 180 ry 0 rz -180 deg; joints [1.363, 71.082, -37.617, 2.471, -33.49, -2.061]
  Call Extruder 0.01786
  MoveL (T18001) to (107.49, 105.16, 19.1) mm, rotated rx 180 ry 0 rz -180 deg; joints [3.241, 71.309, -38.044, 5.895, -33.405, -4.926]
  Call Extruder 0.0573
  MoveL (T18002) to (106.17, 103.84, 19.1) mm, rotated rx 180 ry 0 rz -180 deg; joints [3.241, 71.309, -38.044, 5.895, -33.405, -4.926]
  Call Extruder 0.01786
  MoveL (T18003) to (105.59, 103.84, 19.1) mm, rotated rx 180 ry 0 rz -180 deg; joints [3.241, 71.309, -38.044, 5.895, -33.405, -4.926]
  Call Extruder 0.08219
  MoveL (T18004) to (107.48, 105.73, 19.1) mm, rotated rx 180 ry 0 rz -180 deg; joints [3.351, 66.227, -28.497, 5.466, -37.856, -4.321]
  Call Extruder 0.01786
  MoveL (T18005) to (107.48, 106.32, 19.1) mm, rotated rx 180 ry 0 rz -180 deg; joints [3.351, 66.227, -28.497, 5.466, -37.856, -4.321]
  Call Extruder 0.10744
  MoveL (T18006) to (105.01, 103.84, 19.1) mm, rotated rx 180 ry 0 rz -180 deg; joints [1.409, 66.035, -28.138, 2.294, -37.92, -1.81]
  Call Extruder 0.01786
  MoveL (T18007) to (104.42, 103.84, 19.1) mm, rotated rx 180 ry 0 rz -180 deg; joints [1.409, 66.035, -28.138, 2.294, -37.92, -1.81]
  Call Extruder 0.1327
  MoveL (T18008) to (107.48, 106.9, 19.1) mm, rotated rx 180 ry 0 rz -180 deg; joints [1.407, 66.225, -28.494, 2.299, -37.753, -1.818]
  Call Extruder 0.01087
  MoveL (T18009) to (107.48, 107.25, 19.1) mm, rotated rx 180 ry 0 rz -180 deg; joints [1.407, 66.225, -28.494, 2.299, -37.753, -1.818]
  Call Extruder 0.01602
  MoveL (T18010) to (107.72, 107.72, 19.1) mm, rotated rx 180 ry 0 rz -180 deg; joints [1.365, 66.031, -28.13, 2.222, -37.922, -1.753]
  Call Extruder 0.16825
  MoveL (T18011) to (103.84, 103.84, 19.1) mm, rotated rx 180 ry 0 rz -180 deg; joints [1.365, 66.031, -28.13, 2.222, -37.922, -1.753]
  Call Extruder 0.01786
  MoveL (T18012) to (103.84, 104.42, 19.1) mm, rotated rx 180 ry 0 rz -180 deg; joints [1.365, 66.031, -28.13, 2.222, -37.922, -1.753]
  Call Extruder 0.19454
  MoveL (T18013) to (108.32, 108.9, 19.1) mm, rotated rx 180 ry 0 rz -180 deg; joints [1.365, 66.031, -28.13, 2.222, -37.922, -1.753]
  Call Extruder 0.04092
  MoveL (T18014) to (108.92, 110.09, 19.1) mm, rotated rx 180 ry 0 rz -180 deg; joints [1.365, 66.031, -28.13, 2.222, -37.922, -1.753]
  Call Extruder 0.22084
  MoveL (T18015) to (103.84, 105.01, 19.1) mm, rotated rx 180 ry 0 rz -180 deg; joints [1.365, 66.031, -28.13, 2.222, -37.922, -1.753]
  Call Extruder 0.01786
  MoveL (T18016) to (103.84, 105.59, 19.1) mm, rotated rx 180 ry 0 rz -180 deg; joints [1.319, 71.207, -37.852, 2.399, -33.378, -2.004]
  Call Extruder 0.24714
  MoveL (T18017) to (109.53, 111.27, 19.1) mm, rotated rx 180 ry 0 rz -180 deg; joints [1.319, 71.207, -37.852, 2.399, -33.378, -2.004]
  Call Extruder 0.04092
  MoveL (T18018) to (110.13, 112.46, 19.1) mm, rotated rx 180 ry 0 rz -180 deg; joints [1.319, 71.207, -37.852, 2.399, -33.378, -2.004]
  Call Extruder 0.27344
  MoveL (T18019) to (103.84, 106.17, 19.1) mm, rotated rx 180 ry 0 rz -180 deg; joints [1.319, 71.207, -37.852, 2.399, -33.378, -2.004]
  Call Extruder 0.01786
  MoveL (T18020) to (103.84, 106.75, 19.1) mm, rotated rx 180 ry 0 rz -180 deg; joints [3.282, 71.446, -38.3, 5.986, -33.289, -5.01]
  Call Extruder 0.29974
  MoveL (T18021) to (110.74, 113.64, 19.1) mm, rotated rx 180 ry 0 rz -180 deg; joints [3.282, 71.446, -38.3, 5.986, -33.289, -5.01]
  Call Extruder 0.04092
  MoveL (T18022) to (111.34, 114.83, 19.1) mm, rotated rx 180 ry 0 rz -180 deg; joints [3.398, 66.128, -28.312, 5.531, -37.946, -4.367]
  Call Extruder 0.32604
  MoveL (T18023) to (103.84, 107.33, 19.1) mm, rotated rx 180 ry 0 rz -180 deg; joints [3.398, 66.128, -28.312, 5.531, -37.946, -4.367]
  Call Extruder 0.01786
  MoveL (T18024) to (103.84, 107.91, 19.1) mm, rotated rx 180 ry 0 rz -180 deg; joints [1.366, 65.929, -27.938, 2.219, -38.012, -1.749]
  Call Extruder 0.34996
  MoveL (T18025) to (111.89, 115.96, 19.1) mm, rotated rx 180 ry 0 rz -180 deg; joints [1.366, 65.929, -27.938, 2.219, -38.012, -1.749]
  Call Extruder 0.01786
  MoveL (T18026) to (111.31, 115.96, 19.1) mm, rotated rx 180 ry 0 rz -180 deg; joints [1.366, 65.929, -27.938, 2.219, -38.012, -1.749]
  Call Extruder 0.32471
  MoveL (T18027) to (103.84, 108.49, 19.1) mm, rotated rx 180 ry 0 rz -180 deg; joints [1.365, 66.016, -28.101, 2.221, -37.936, -1.752]
  Call Extruder 0.01786
  MoveL (T18028) to (103.84, 109.07, 19.1) mm, rotated rx 180 ry 0 rz -180 deg; joints [1.365, 66.016, -28.101, 2.221, -37.936, -1.752]
  Call Extruder 0.29945
  MoveL (T18029) to (110.73, 115.96, 19.1) mm, rotated rx 180 ry 0 rz -180 deg; joints [1.365, 66.016, -28.101, 2.221, -37.936, -1.752]
  Call Extruder 0.01786
  MoveL (T18030) to (110.15, 115.96, 19.1) mm, rotated rx 180 ry 0 rz -180 deg; joints [1.332, 65.823, -27.74, 2.16, -38.103, -1.7]
  Call Extruder 0.2742
  MoveL (T18031) to (103.84, 109.65, 19.1) mm, rotated rx 180 ry 0 rz -180 deg; joints [1.332, 65.823, -27.74, 2.16, -38.103, -1.7]
  Call Extruder 0.01786
  MoveL (T18032) to (103.84, 110.23, 19.1) mm, rotated rx 180 ry 0 rz -180 deg; joints [1.332, 65.823, -27.74, 2.16, -38.103, -1.7]
  Call Extruder 0.24895
  MoveL (T18033) to (109.57, 115.96, 19.1) mm, rotated rx 180 ry 0 rz -180 deg; joints [1.332, 65.823, -27.74, 2.16, -38.103, -1.7]
  Call Extruder 0.01786
  MoveL (T18034) to (108.99, 115.96, 19.1) mm, rotated rx 180 ry 0 rz -180 deg; joints [1.332, 65.823, -27.74, 2.16, -38.103, -1.7]
  Call Extruder 0.22369
  MoveL (T18035) to (103.84, 110.82, 19.1) mm, rotated rx 180 ry 0 rz -180 deg; joints [1.332, 65.823, -27.74, 2.16, -38.103, -1.7]
  Call Extruder 0.01786
  MoveL (T18036) to (103.84, 111.4, 19.1) mm, rotated rx 180 ry 0 rz -180 deg; joints [1.323, 65.823, -27.739, 2.145, -38.103, -1.688]
  Call Extruder 0.19844
  MoveL (T18037) to (108.41, 115.96, 19.1) mm, rotated rx 180 ry 0 rz -180 deg; joints [1.323, 65.823, -27.739, 2.145, -38.103, -1.688]
  Call Extruder 0.01786
  MoveL (T18038) to (107.83, 115.96, 19.1) mm, rotated rx 180 ry 0 rz -180 deg; joints [1.276, 71.333, -38.088, 2.326, -33.266, -1.946]
  Call Extruder 0.17318
  MoveL (T18039) to (103.84, 111.98, 19.1) mm, rotated rx 180 ry 0 rz -180 deg; joints [1.276, 71.333, -38.088, 2.326, -33.266, -1.946]
  Call Extruder 0.01786
  MoveL (T18040) to (103.84, 112.56, 19.1) mm, rotated rx 180 ry 0 rz -180 deg; joints [1.276, 71.333, -38.088, 2.326, -33.266, -1.946]
  Call Extruder 0.1616
  MoveL (T18041) to (107.56, 116.28, 19.1) mm, rotated rx 180 ry 0 rz -180 deg; joints [1.276, 71.333, -38.088, 2.326, -33.266, -1.946]
  Call Extruder 0.01786
  MoveL (T18042) to (107.56, 116.86, 19.1) mm, rotated rx 180 ry 0 rz -180 deg; joints [3.322, 71.583, -38.559, 6.079, -33.172, -5.094]
  Call Extruder 0.1616
  MoveL (T18043) to (103.84, 113.14, 19.1) mm, rotated rx 180 ry 0 rz -180 deg; joints [3.322, 71.583, -38.559, 6.079, -33.172, -5.094]
  Call Extruder 0.01786
  MoveL (T18044) to (103.84, 113.72, 19.1) mm, rotated rx 180 ry 0 rz -180 deg; joints [3.322, 71.583, -38.559, 6.079, -33.172, -5.094]
  Call Extruder 0.1616
  MoveL (T18045) to (107.56, 117.44, 19.1) mm, rotated rx 180 ry 0 rz -180 deg; joints [3.322, 71.583, -38.559, 6.079, -33.172, -5.094]
  Call Extruder 0.01786
  MoveL (T18046) to (107.56, 118.02, 19.1) mm, rotated rx 180 ry 0 rz -180 deg; joints [3.445, 66.03, -28.128, 5.596, -38.035, -4.413]
  Call Extruder 0.1616
  MoveL (T18047) to (103.84, 114.3, 19.1) mm, rotated rx 180 ry 0 rz -180 deg; joints [3.445, 66.03, -28.128, 5.596, -38.035, -4.413]
  Call Extruder 0.01786
  MoveL (T18048) to (103.84, 114.88, 19.1) mm, rotated rx 180 ry 0 rz -180 deg; joints [3.445, 66.03, -28.128, 5.596, -38.035, -4.413]
  Call Extruder 0.1616
  MoveL (T18049) to (107.56, 118.6, 19.1) mm, rotated rx 180 ry 0 rz -180 deg; joints [1.339, 65.824, -27.741, 2.17, -38.103, -1.708]
  Call Extruder 0.01786
  MoveL (T18050) to (107.56, 119.18, 19.1) mm, rotated rx 180 ry 0 rz -180 deg; joints [1.339, 65.824, -27.741, 2.17, -38.103, -1.708]
  Call Extruder 0.16957
  MoveL (T18051) to (103.66, 115.28, 19.1) mm, rotated rx 180 ry 0 rz -180 deg; joints [1.326, 65.838, -27.768, 2.149, -38.09, -1.692]
  Set speed (45.0 mm/s)
  Call Extruder -1.6
  MoveL (T18052) to (103.66, 115.28, 19.1) mm, rotated rx 180 ry 0 rz -180 deg; joints [1.326, 65.838, -27.768, 2.149, -38.09, -1.692]
  Set speed (120.0 mm/s)
  MoveL (T18053) to (103.66, 115.28, 19.1) mm, rotated rx 180 ry 0 rz -180 deg; joints [1.326, 65.838, -27.768, 2.149, -38.09, -1.692]
  Call Extruder -0.38
  MoveL (T18054) to (104.42, 116.03, 19.1) mm, rotated rx 180 ry 0 rz -180 deg; joints [1.326, 65.838, -27.768, 2.149, -38.09, -1.692]
  Set speed (45.0 mm/s)
  Call Extruder -0.02
  MoveL (T18055) to (104.42, 116.03, 19.1) mm, rotated rx 180 ry 0 rz -180 deg; joints [1.326, 65.838, -27.768, 2.149, -38.09, -1.692]
  Set speed (150.0 mm/s)
  MoveL (T18056) to (104.42, 116.03, 21.1) mm, rotated rx 180 ry 0 rz -180 deg; joints [1.326, 65.838, -27.768, 2.149, -38.09, -1.692]
  MoveL (T18057) to (117.77, 105.57, 21.1) mm, rotated rx 180 ry 0 rz -180 deg; joints [1.326, 65.838, -27.768, 2.149, -38.09, -1.692]
  MoveL (T18058) to (117.77, 105.57, 19.1) mm, rotated rx 180 ry 0 rz -180 deg; joints [1.326, 65.838, -27.768, 2.149, -38.09, -1.692]
  Set speed (40.0 mm/s)
  Call Extruder 2.0
  MoveL (T18059) to (117.77, 105.57, 19.1) mm, rotated rx 180 ry 0 rz -180 deg; joints [1.326, 65.838, -27.768, 2.149, -38.09, -1.692]
  Call Extruder 0.14703
  MoveL (T18060) to (121.16, 108.96, 19.1) mm, rotated rx 180 ry 0 rz -180 deg; joints [1.326, 65.838, -27.768, 2.149, -38.09, -1.692]
  Call Extruder 0.01786
  MoveL (T18061) to (121.16, 109.54, 19.1) mm, rotated rx 180 ry 0 rz -180 deg; joints [1.326, 65.838, -27.768, 2.149, -38.09, -1.692]
  Call Extruder 0.13907
  MoveL (T18062) to (117.96, 106.34, 19.1) mm, rotated rx 180 ry 0 rz -180 deg; joints [1.326, 65.838, -27.768, 2.149, -38.09, -1.692]
  Call Extruder 0.01786
  MoveL (T18063) to (117.96, 106.92, 19.1) mm, rotated rx 180 ry 0 rz -180 deg; joints [1.323, 65.823, -27.739, 2.145, -38.103, -1.688]
  Call Extruder 0.13907
  MoveL (T18064) to (121.16, 110.12, 19.1) mm, rotated rx 180 ry 0 rz -180 deg; joints [1.321, 66.058, -28.18, 2.151, -37.897, -1.697]
  Call Extruder 0.01786
  MoveL (T18065) to (121.16, 110.7, 19.1) mm, rotated rx 180 ry 0 rz -180 deg; joints [1.321, 66.058, -28.18, 2.151, -37.897, -1.697]
  Call Extruder 0.13907
  MoveL (T18066) to (117.96, 107.5, 19.1) mm, rotated rx 180 ry 0 rz -180 deg; joints [1.321, 66.058, -28.18, 2.151, -37.897, -1.697]
  Call Extruder 0.01786
  MoveL (T18067) to (117.96, 108.08, 19.1) mm, rotated rx 180 ry 0 rz -180 deg; joints [1.321, 66.058, -28.18, 2.151, -37.897, -1.697]
  Call Extruder 0.13907
  MoveL (T18068) to (121.16, 111.28, 19.1) mm, rotated rx 180 ry 0 rz -180 deg; joints [1.321, 66.058, -28.18, 2.151, -37.897, -1.697]
  Call Extruder 0.01786
  MoveL (T18069) to (121.16, 111.86, 19.1) mm, rotated rx 180 ry 0 rz -180 deg; joints [1.321, 66.058, -28.18, 2.151, -37.897, -1.697]
  Call Extruder 0.13907
  MoveL (T18070) to (117.96, 108.66, 19.1) mm, rotated rx 180 ry 0 rz -180 deg; joints [1.321, 66.058, -28.18, 2.151, -37.897, -1.697]
  Call Extruder 0.01786
  MoveL (T18071) to (117.96, 109.24, 19.1) mm, rotated rx 180 ry 0 rz -180 deg; joints [1.707, 65.897, -28.285, 2.795, -37.645, -2.214]
  Call Extruder 0.13907
  MoveL (T18072) to (121.16, 112.44, 19.1) mm, rotated rx 180 ry 0 rz -180 deg; joints [1.707, 66.133, -28.32, 2.782, -37.845, -2.198]
  Call Extruder 0.01786
  MoveL (T18073) to (121.16, 113.02, 19.1) mm, rotated rx 180 ry 0 rz -180 deg; joints [1.707, 66.133, -28.32, 2.782, -37.845, -2.198]
  Call Extruder 0.15905
  MoveL (T18074) to (117.5, 109.36, 19.1) mm, rotated rx 180 ry 0 rz -180 deg; joints [1.707, 66.133, -28.32, 2.782, -37.845, -2.198]
  Call Extruder 0.01786
  MoveL (T18075) to (116.92, 109.36, 19.1) mm, rotated rx 180 ry 0 rz -180 deg; joints [1.707, 66.133, -28.32, 2.782, -37.845, -2.198]
  Call Extruder 0.1843
  MoveL (T18076) to (121.16, 113.6, 19.1) mm, rotated rx 180 ry 0 rz -180 deg; joints [1.707, 66.133, -28.32, 2.782, -37.845, -2.198]
  Call Extruder 0.01786
  MoveL (T18077) to (121.16, 114.19, 19.1) mm, rotated rx 180 ry 0 rz -180 deg; joints [1.707, 66.133, -28.32, 2.782, -37.845, -2.198]
  Call Extruder 0.20956
  MoveL (T18078) to (116.33, 109.36, 19.1) mm, rotated rx 180 ry 0 rz -180 deg; joints [1.707, 66.133, -28.32, 2.782, -37.845, -2.198]
  Call Extruder 0.01786
  MoveL (T18079) to (115.75, 109.36, 19.1) mm, rotated rx 180 ry 0 rz -180 deg; joints [1.707, 66.133, -28.32, 2.782, -37.845, -2.198]
  Call Extruder 0.23481
  MoveL (T18080) to (121.16, 114.77, 19.1) mm, rotated rx 180 ry 0 rz -180 deg; joints [1.707, 66.133, -28.32, 2.782, -37.845, -2.198]
  Call Extruder 0.01786
  MoveL (T18081) to (121.16, 115.35, 19.1) mm, rotated rx 180 ry 0 rz -180 deg; joints [1.707, 66.133, -28.32, 2.782, -37.845, -2.198]
  Call Extruder 0.26007
  MoveL (T18082) to (115.17, 109.36, 19.1) mm, rotated rx 180 ry 0 rz -180 deg; joints [1.442, 66.115, -28.288, 2.35, -37.851, -1.856]
  Call Extruder 0.01786
  MoveL (T18083) to (114.59, 109.36, 19.1) mm, rotated rx 180 ry 0 rz -180 deg; joints [1.442, 66.115, -28.288, 2.35, -37.851, -1.856]
  Call Extruder 0.28532
  MoveL (T18084) to (121.16, 115.93, 19.1) mm, rotated rx 180 ry 0 rz -180 deg; joints [1.657, 66.131, -28.316, 2.702, -37.845, -2.134]
  Call Extruder 0.01786
  MoveL (T18085) to (121.16, 116.51, 19.1) mm, rotated rx 180 ry 0 rz -180 deg; joints [1.657, 66.131, -28.316, 2.702, -37.845, -2.134]
  Call Extruder 0.31058
  MoveL (T18086) to (114.01, 109.36, 19.1) mm, rotated rx 180 ry 0 rz -180 deg; joints [1.657, 66.131, -28.316, 2.702, -37.845, -2.134]
  Call Extruder 0.01786
  MoveL (T18087) to (113.43, 109.36, 19.1) mm, rotated rx 180 ry 0 rz -180 deg; joints [1.679, 66.153, -28.359, 2.738, -37.826, -2.163]
  Call Extruder 0.33583
  MoveL (T18088) to (121.16, 117.09, 19.1) mm, rotated rx 180 ry 0 rz -180 deg; joints [1.679, 66.153, -28.359, 2.738, -37.826, -2.163]
  Call Extruder 0.01786
  MoveL (T18089) to (121.16, 117.67, 19.1) mm, rotated rx 180 ry 0 rz -180 deg; joints [1.679, 66.153, -28.359, 2.738, -37.826, -2.163]
  Call Extruder 0.31968
  MoveL (T18090) to (113.8, 110.32, 19.1) mm, rotated rx 180 ry 0 rz -180 deg; joints [1.679, 66.153, -28.359, 2.738, -37.826, -2.163]
  Call Extruder 0.04109
  MoveL (T18091) to (114.41, 111.51, 19.1) mm, rotated rx 180 ry 0 rz -180 deg; joints [1.743, 66.315, -28.662, 2.851, -37.687, -2.257]
  Call Extruder 0.29321
  MoveL (T18092) to (121.16, 118.25, 19.1) mm, rotated rx 180 ry 0 rz -180 deg; joints [1.743, 66.315, -28.662, 2.851, -37.687, -2.257]
  Call Extruder 0.01786
  MoveL (T18093) to (121.16, 118.83, 19.1) mm, rotated rx 180 ry 0 rz -180 deg; joints [1.743, 66.315, -28.662, 2.851, -37.687, -2.257]
  Call Extruder 0.26675
  MoveL (T18094) to (115.02, 112.7, 19.1) mm, rotated rx 180 ry 0 rz -180 deg; joints [1.821, 66.141, -28.336, 2.968, -37.842, -2.345]
  Call Extruder 0.04109
  MoveL (T18095) to (115.63, 113.89, 19.1) mm, rotated rx 180 ry 0 rz -180 deg; joints [1.941, 66.15, -28.354, 3.165, -37.839, -2.5]
  Call Extruder 0.24028
  MoveL (T18096) to (121.16, 119.41, 19.1) mm, rotated rx 180 ry 0 rz -180 deg; joints [1.941, 66.15, -28.354, 3.165, -37.839, -2.5]
  Call Extruder 0.01786
  MoveL (T18097) to (121.16, 119.99, 19.1) mm, rotated rx 180 ry 0 rz -180 deg; joints [1.941, 66.15, -28.354, 3.165, -37.839, -2.5]
  Call Extruder 0.21381
  MoveL (T18098) to (116.24, 115.08, 19.1) mm, rotated rx 180 ry 0 rz -180 deg; joints [3.239, 69.802, -35.211, 5.692, -34.723, -4.683]
  Call Extruder 0.04109
  MoveL (T18099) to (116.85, 116.27, 19.1) mm, rotated rx 180 ry 0 rz -180 deg; joints [3.239, 69.802, -35.211, 5.692, -34.723, -4.683]
  Call Extruder 0.18734
  MoveL (T18100) to (121.16, 120.58, 19.1) mm, rotated rx 180 ry 0 rz -180 deg; joints [3.239, 69.802, -35.211, 5.692, -34.723, -4.683]
  Call Extruder 0.01786
  MoveL (T18101) to (121.16, 121.16, 19.1) mm, rotated rx 180 ry 0 rz -180 deg; joints [3.232, 70.133, -35.833, 5.722, -34.433, -4.725]
  Call Extruder 0.16087
  MoveL (T18102) to (117.45, 117.45, 19.1) mm, rotated rx 180 ry 0 rz -180 deg; joints [3.232, 70.133, -35.833, 5.722, -34.433, -4.725]
  Call Extruder 0.02137
  MoveL (T18103) to (117.77, 118.07, 19.1) mm, rotated rx 180 ry 0 rz -180 deg; joints [3.232, 70.133, -35.833, 5.722, -34.433, -4.725]
  Call Extruder 0.00857
  MoveL (T18104) to (117.77, 118.35, 19.1) mm, rotated rx 180 ry 0 rz -180 deg; joints [2.845, 71.149, -37.743, 5.158, -33.513, -4.304]
  Call Extruder 0.12185
  MoveL (T18105) to (120.58, 121.16, 19.1) mm, rotated rx 180 ry 0 rz -180 deg; joints [2.845, 71.149, -37.743, 5.158, -33.513, -4.304]
  Call Extruder 0.01786
  MoveL (T18106) to (119.99, 121.16, 19.1) mm, rotated rx 180 ry 0 rz -180 deg; joints [3.211, 71.208, -37.852, 5.826, -33.492, -4.864]
  Call Extruder 0.09659
  MoveL (T18107) to (117.77, 118.93, 19.1) mm, rotated rx 180 ry 0 rz -180 deg; joints [3.211, 71.208, -37.852, 5.826, -33.492, -4.864]
  Call Extruder 0.01786
  MoveL (T18108) to (117.77, 119.52, 19.1) mm, rotated rx 180 ry 0 rz -180 deg; joints [3.211, 71.208, -37.852, 5.826, -33.492, -4.864]
  Call Extruder 0.07134
  MoveL (T18109) to (119.41, 121.16, 19.1) mm, rotated rx 180 ry 0 rz -180 deg; joints [1.893, 67.277, -30.468, 3.158, -36.85, -2.528]
  Call Extruder 0.01786
  MoveL (T18110) to (118.83, 121.16, 19.1) mm, rotated rx 180 ry 0 rz -180 deg; joints [1.893, 67.277, -30.468, 3.158, -36.85, -2.528]
  Call Extruder 0.04608
  MoveL (T18111) to (117.77, 120.1, 19.1) mm, rotated rx 180 ry 0 rz -180 deg; joints [1.895, 67.14, -30.211, 3.152, -36.97, -2.519]
  Call Extruder 0.00206
  MoveL (T18112) to (117.77, 120.16, 19.1) mm, rotated rx 180 ry 0 rz -180 deg; joints [1.895, 67.14, -30.211, 3.152, -36.97, -2.519]
  Call Extruder 0.0158
  MoveL (T18113) to (117.26, 120.16, 19.1) mm, rotated rx 180 ry 0 rz -180 deg; joints [2.319, 66.184, -28.416, 3.784, -37.828, -2.99]
  Call Extruder 0.04317
  MoveL (T18114) to (118.25, 121.16, 19.1) mm, rotated rx 180 ry 0 rz -180 deg; joints [2.319, 66.184, -28.416, 3.784, -37.828, -2.99]
  Call Extruder 0.01786
  MoveL (T18115) to (117.67, 121.16, 19.1) mm, rotated rx 180 ry 0 rz -180 deg; joints [2.319, 66.184, -28.416, 3.784, -37.828, -2.99]
  Call Extruder 0.04317
  MoveL (T18116) to (116.68, 120.16, 19.1) mm, rotated rx 180 ry 0 rz -180 deg; joints [2.44, 66.196, -28.439, 3.981, -37.824, -3.146]
  Call Extruder 0.01786
  MoveL (T18117) to (116.1, 120.16, 19.1) mm, rotated rx 180 ry 0 rz -180 deg; joints [2.44, 66.196, -28.439, 3.981, -37.824, -3.146]
  Call Extruder 0.04317
  MoveL (T18118) to (117.09, 121.16, 19.1) mm, rotated rx 180 ry 0 rz -180 deg; joints [2.44, 66.196, -28.439, 3.981, -37.824, -3.146]
  Call Extruder 0.01786
  MoveL (T18119) to (116.51, 121.16, 19.1) mm, rotated rx 180 ry 0 rz -180 deg; joints [3.266, 68.476, -32.72, 5.578, -35.885, -4.524]
  Call Extruder 0.04317
  MoveL (T18120) to (115.52, 120.16, 19.1) mm, rotated rx 180 ry 0 rz -180 deg; joints [3.266, 68.476, -32.72, 5.578, -35.885, -4.524]
  Call Extruder 0.01786
  MoveL (T18121) to (114.93, 120.16, 19.1) mm, rotated rx 180 ry 0 rz -180 deg; joints [3.26, 68.789, -33.309, 5.604, -35.61, -4.561]
  Call Extruder 0.04317
  MoveL (T18122) to (115.93, 121.16, 19.1) mm, rotated rx 180 ry 0 rz -180 deg; joints [3.26, 68.789, -33.309, 5.604, -35.61, -4.561]
  Call Extruder 0.01786
  MoveL (T18123) to (115.35, 121.16, 19.1) mm, rotated rx 180 ry 0 rz -180 deg; joints [2.685, 70.221, -35.998, 4.766, -34.315, -3.939]
  Call Extruder 0.04317
  MoveL (T18124) to (114.35, 120.16, 19.1) mm, rotated rx 180 ry 0 rz -180 deg; joints [2.685, 70.221, -35.998, 4.766, -34.315, -3.939]
  Call Extruder 0.01786
  MoveL (T18125) to (113.77, 120.16, 19.1) mm, rotated rx 180 ry 0 rz -180 deg; joints [2.754, 70.44, -36.411, 4.913, -34.127, -4.07]
  Call Extruder 0.04317
  MoveL (T18126) to (114.77, 121.16, 19.1) mm, rotated rx 180 ry 0 rz -180 deg; joints [2.754, 70.44, -36.411, 4.913, -34.127, -4.07]
  Call Extruder 0.01786
  MoveL (T18127) to (114.18, 121.16, 19.1) mm, rotated rx 180 ry 0 rz -180 deg; joints [2.754, 70.44, -36.411, 4.913, -34.127, -4.07]
  Call Extruder 0.04317
  MoveL (T18128) to (113.19, 120.16, 19.1) mm, rotated rx 180 ry 0 rz -180 deg; joints [2.762, 70.503, -36.528, 4.934, -34.073, -4.09]
  Call Extruder 0.01786
  MoveL (T18129) to (112.61, 120.16, 19.1) mm, rotated rx 180 ry 0 rz -180 deg; joints [2.762, 70.503, -36.528, 4.934, -34.073, -4.09]
  Call Extruder 0.04317
  MoveL (T18130) to (113.6, 121.16, 19.1) mm, rotated rx 180 ry 0 rz -180 deg; joints [2.762, 70.503, -36.528, 4.934, -34.073, -4.09]
  Call Extruder 0.01786
  MoveL (T18131) to (113.02, 121.16, 19.1) mm, rotated rx 180 ry 0 rz -180 deg; joints [2.756, 70.887, -37.249, 4.966, -33.737, -4.133]
  Call Extruder 0.04317
  MoveL (T18132) to (112.03, 120.16, 19.1) mm, rotated rx 180 ry 0 rz -180 deg; joints [2.756, 70.887, -37.249, 4.966, -33.737, -4.133]
  Call Extruder 0.01786
  MoveL (T18133) to (111.45, 120.16, 19.1) mm, rotated rx 180 ry 0 rz -180 deg; joints [2.756, 70.887, -37.249, 4.966, -33.737, -4.133]
  Call Extruder 0.04317
  MoveL (T18134) to (112.44, 121.16, 19.1) mm, rotated rx 180 ry 0 rz -180 deg; joints [2.756, 70.887, -37.249, 4.966, -33.737, -4.133]
  Call Extruder 0.01786
  MoveL (T18135) to (111.86, 121.16, 19.1) mm, rotated rx 180 ry 0 rz -180 deg; joints [2.633, 71.177, -37.794, 4.778, -33.474, -3.988]
  Call Extruder 0.04317
  MoveL (T18136) to (110.87, 120.16, 19.1) mm, rotated rx 180 ry 0 rz -180 deg; joints [2.633, 71.177, -37.794, 4.778, -33.474, -3.988]
  Call Extruder 0.01786
  MoveL (T18137) to (110.29, 120.16, 19.1) mm, rotated rx 180 ry 0 rz -180 deg; joints [2.633, 71.177, -37.794, 4.778, -33.474, -3.988]
  Call Extruder 0.04317
  MoveL (T18138) to (111.28, 121.16, 19.1) mm, rotated rx 180 ry 0 rz -180 deg; joints [2.633, 71.177, -37.794, 4.778, -33.474, -3.988]
  Call Extruder 0.01786
  MoveL (T18139) to (110.7, 121.16, 19.1) mm, rotated rx 180 ry 0 rz -180 deg; joints [2.633, 71.177, -37.794, 4.778, -33.474, -3.988]
  Call Extruder 0.04317
  MoveL (T18140) to (109.71, 120.16, 19.1) mm, rotated rx 180 ry 0 rz -180 deg; joints [2.633, 71.177, -37.794, 4.778, -33.474, -3.988]
  Call Extruder 0.01786
  MoveL (T18141) to (109.12, 120.16, 19.1) mm, rotated rx 180 ry 0 rz -180 deg; joints [2.633, 71.177, -37.794, 4.778, -33.474, -3.988]
  Call Extruder 0.04317
  MoveL (T18142) to (110.12, 121.16, 19.1) mm, rotated rx 180 ry 0 rz -180 deg; joints [2.712, 70.962, -37.392, 4.895, -33.667, -4.077]
  Call Extruder 0.01786
  MoveL (T18143) to (109.54, 121.16, 19.1) mm, rotated rx 180 ry 0 rz -180 deg; joints [2.714, 70.783, -37.055, 4.881, -33.824, -4.057]
  Call Extruder 0.05113
  MoveL (T18144) to (108.36, 119.98, 19.1) mm, rotated rx 180 ry 0 rz -180 deg; joints [2.714, 70.783, -37.055, 4.881, -33.824, -4.057]
  Set speed (150.0 mm/s)
  MoveL (T18145) to (109.14, 121.34, 19.1) mm, rotated rx 180 ry 0 rz -180 deg; joints [2.592, 71.113, -37.676, 4.697, -33.527, -3.918]
  Set speed (40.0 mm/s)
  MoveL (T18146) to (109.14, 121.34, 19.1) mm, rotated rx 180 ry 0 rz -180 deg; joints [2.532, 71.105, -37.66, 4.587, -33.53, -3.826]
  Call Extruder 0.05113
  MoveL (T18147) to (107.96, 120.16, 19.1) mm, rotated rx 180 ry 0 rz -180 deg; joints [2.532, 71.105, -37.66, 4.587, -33.53, -3.826]
  Call Extruder 0.01234
  MoveL (T18148) to (107.56, 120.16, 19.1) mm, rotated rx 180 ry 0 rz -180 deg; joints [2.717, 70.605, -36.72, 4.866, -33.981, -4.038]
  Call Extruder 0.01234
  MoveL (T18149) to (107.56, 119.76, 19.1) mm, rotated rx 180 ry 0 rz -180 deg; joints [2.717, 70.605, -36.72, 4.866, -33.981, -4.038]
  Call Extruder 0.1616
  MoveL (T18150) to (103.84, 116.04, 19.1) mm, rotated rx 180 ry 0 rz -180 deg; joints [2.717, 70.605, -36.72, 4.866, -33.981, -4.038]
  Call Extruder 0.01786
  MoveL (T18151) to (103.84, 116.62, 19.1) mm, rotated rx 180 ry 0 rz -180 deg; joints [2.719, 70.522, -36.564, 4.859, -34.054, -4.029]
  Call Extruder 0.19697
  MoveL (T18152) to (108.38, 121.16, 19.1) mm, rotated rx 180 ry 0 rz -180 deg; joints [2.719, 70.522, -36.564, 4.859, -34.054, -4.029]
  Call Extruder 0.01786
  MoveL (T18153) to (107.79, 121.16, 19.1) mm, rotated rx 180 ry 0 rz -180 deg; joints [2.719, 70.522, -36.564, 4.859, -34.054, -4.029]
  Call Extruder 0.17171
  MoveL (T18154) to (103.84, 117.21, 19.1) mm, rotated rx 180 ry 0 rz -180 deg; joints [2.717, 70.506, -36.534, 4.854, -34.067, -4.024]
  Call Extruder 0.01786
  MoveL (T18155) to (103.84, 117.79, 19.1) mm, rotated rx 180 ry 0 rz -180 deg; joints [2.717, 70.506, -36.534, 4.854, -34.067, -4.024]
  Call Extruder 0.14646
  MoveL (T18156) to (107.21, 121.16, 19.1) mm, rotated rx 180 ry 0 rz -180 deg; joints [2.717, 70.506, -36.534, 4.854, -34.067, -4.024]
  Call Extruder 0.01786
  MoveL (T18157) to (106.63, 121.16, 19.1) mm, rotated rx 180 ry 0 rz -180 deg; joints [2.717, 70.506, -36.534, 4.854, -34.067, -4.024]
  Call Extruder 0.1212
  MoveL (T18158) to (103.84, 118.37, 19.1) mm, rotated rx 180 ry 0 rz -180 deg; joints [2.705, 70.468, -36.463, 4.829, -34.1, -4.001]
  Call Extruder 0.01786
  MoveL (T18159) to (103.84, 118.95, 19.1) mm, rotated rx 180 ry 0 rz -180 deg; joints [2.471, 71.097, -37.645, 4.476, -33.533, -3.734]
  Call Extruder 0.09595
  MoveL (T18160) to (106.05, 121.16, 19.1) mm, rotated rx 180 ry 0 rz -180 deg; joints [2.471, 71.097, -37.645, 4.476, -33.533, -3.734]
  Call Extruder 0.01786
  MoveL (T18161) to (105.47, 121.16, 19.1) mm, rotated rx 180 ry 0 rz -180 deg; joints [2.471, 71.097, -37.645, 4.476, -33.533, -3.734]
  Call Extruder 0.07069
  MoveL (T18162) to (103.84, 119.53, 19.1) mm, rotated rx 180 ry 0 rz -180 deg; joints [2.41, 71.09, -37.631, 4.366, -33.535, -3.641]
  Call Extruder 0.01786
  MoveL (T18163) to (103.84, 120.11, 19.1) mm, rotated rx 180 ry 0 rz -180 deg; joints [2.41, 71.09, -37.631, 4.366, -33.535, -3.641]
  Call Extruder 0.04544
  MoveL (T18164) to (104.89, 121.16, 19.1) mm, rotated rx 180 ry 0 rz -180 deg; joints [2.676, 70.376, -36.29, 4.767, -34.178, -3.947]
  Call Extruder 0.01786
  MoveL (T18165) to (104.31, 121.16, 19.1) mm, rotated rx 180 ry 0 rz -180 deg; joints [2.676, 70.376, -36.29, 4.767, -34.178, -3.947]
  Call Extruder 0.02815
  MoveL (T18166) to (103.66, 120.51, 19.1) mm, rotated rx 180 ry 0 rz -180 deg; joints [2.676, 70.376, -36.29, 4.767, -34.178, -3.947]
  Set speed (45.0 mm/s)
  Call Extruder -1.6
  MoveL (T18167) to (103.66, 120.51, 19.1) mm, rotated rx 180 ry 0 rz -180 deg; joints [2.647, 70.284, -36.118, 4.706, -34.257, -3.892]
  Set speed (120.0 mm/s)
  MoveL (T18168) to (103.66, 120.51, 19.1) mm, rotated rx 180 ry 0 rz -180 deg; joints [2.647, 70.284, -36.118, 4.706, -34.257, -3.892]
  Call Extruder -0.3262
  MoveL (T18169) to (104.31, 121.16, 19.1) mm, rotated rx 180 ry 0 rz -180 deg; joints [2.647, 70.284, -36.118, 4.706, -34.257, -3.892]
  Call Extruder -0.0538
  MoveL (T18170) to (104.46, 121.16, 19.1) mm, rotated rx 180 ry 0 rz -180 deg; joints [2.647, 70.284, -36.118, 4.706, -34.257, -3.892]
  Set speed (45.0 mm/s)
  Call Extruder -0.02
  MoveL (T18171) to (104.46, 121.16, 19.1) mm, rotated rx 180 ry 0 rz -180 deg; joints [2.35, 71.082, -37.617, 4.256, -33.538, -3.549]
  Set speed (150.0 mm/s)
  MoveL (T18172) to (104.46, 121.16, 21.1) mm, rotated rx 180 ry 0 rz -180 deg; joints [2.35, 71.082, -37.617, 4.256, -33.538, -3.549]
  MoveL (T18173) to (109.4, 105.47, 21.1) mm, rotated rx 180 ry 0 rz -180 deg; joints [2.289, 71.075, -37.603, 4.145, -33.541, -3.457]
  MoveL (T18174) to (109.4, 105.47, 19.3) mm, rotated rx 180 ry 0 rz -180 deg; joints [2.289, 71.075, -37.603, 4.145, -33.541, -3.457]
  Set speed (40.0 mm/s)
  Call Extruder 2.0
  MoveL (T18175) to (109.4, 105.47, 19.3) mm, rotated rx 180 ry 0 rz -180 deg; joints [2.289, 71.075, -37.603, 4.145, -33.541, -3.457]
  Call Extruder 0.25145
  MoveL (T18176) to (117.65, 105.47, 19.3) mm, rotated rx 180 ry 0 rz -180 deg; joints [2.618, 70.193, -35.946, 4.644, -34.335, -3.838]
  Call Extruder 0.10939
  MoveL (T18177) to (117.65, 109.06, 19.3) mm, rotated rx 180 ry 0 rz -180 deg; joints [2.618, 70.193, -35.946, 4.644, -34.335, -3.838]
  Call Extruder 0.14732
  MoveL (T18178) to (112.81, 109.06, 19.3) mm, rotated rx 180 ry 0 rz -180 deg; joints [2.588, 70.102, -35.775, 4.584, -34.412, -3.784]
  Call Extruder 0.31102
  MoveL (T18179) to (117.47, 118.15, 19.3) mm, rotated rx 180 ry 0 rz -180 deg; joints [2.588, 70.102, -35.775, 4.584, -34.412, -3.784]
  Call Extruder 0.05209
  MoveL (T18180) to (117.47, 119.86, 19.3) mm, rotated rx 180 ry 0 rz -180 deg; joints [2.588, 70.102, -35.775, 4.584, -34.412, -3.784]
  Call Extruder 0.29244
  MoveL (T18181) to (107.87, 119.86, 19.3) mm, rotated rx 180 ry 0 rz -180 deg; joints [2.228, 71.068, -37.589, 4.035, -33.544, -3.365]
  Call Extruder 0.10939
  MoveL (T18182) to (107.87, 116.27, 19.3) mm, rotated rx 180 ry 0 rz -180 deg; joints [2.228, 71.068, -37.589, 4.035, -33.544, -3.365]
  Call Extruder 0.13869
  MoveL (T18183) to (112.42, 116.27, 19.3) mm, rotated rx 180 ry 0 rz -180 deg; joints [2.168, 71.061, -37.576, 3.924, -33.546, -3.272]
  Call Extruder 0.31084
  MoveL (T18184) to (107.78, 107.18, 19.3) mm, rotated rx 180 ry 0 rz -180 deg; joints [2.168, 71.061, -37.576, 3.924, -33.546, -3.272]
  Call Extruder 0.05206
  MoveL (T18185) to (107.78, 105.47, 19.3) mm, rotated rx 180 ry 0 rz -180 deg; joints [2.559, 70.012, -35.605, 4.523, -34.49, -3.73]
  Call Extruder 0.04735
  MoveL (T18186) to (109.34, 105.47, 19.3) mm, rotated rx 180 ry 0 rz -180 deg; joints [2.559, 70.012, -35.605, 4.523, -34.49, -3.73]
  Set speed (150.0 mm/s)
  MoveL (T18187) to (109, 105.88, 19.3) mm, rotated rx 180 ry 0 rz -180 deg; joints [2.559, 70.012, -35.605, 4.523, -34.49, -3.73]
  Set speed (40.0 mm/s)
  MoveL (T18188) to (109, 105.88, 19.3) mm, rotated rx 180 ry 0 rz -180 deg; joints [2.559, 70.012, -35.605, 4.523, -34.49, -3.73]
  Call Extruder 0.25124
  MoveL (T18189) to (117.24, 105.88, 19.3) mm, rotated rx 180 ry 0 rz -180 deg; joints [2.53, 69.921, -35.435, 4.462, -34.567, -3.677]
  Call Extruder 0.08459
  MoveL (T18190) to (117.24, 108.65, 19.3) mm, rotated rx 180 ry 0 rz -180 deg; joints [2.53, 69.921, -35.435, 4.462, -34.567, -3.677]
  Call Extruder 0.1552
  MoveL (T18191) to (112.15, 108.65, 19.3) mm, rotated rx 180 ry 0 rz -180 deg; joints [2.53, 69.921, -35.435, 4.462, -34.567, -3.677]
  Call Extruder 0.32831
  MoveL (T18192) to (117.06, 118.25, 19.3) mm, rotated rx 180 ry 0 rz -180 deg; joints [2.107, 71.054, -37.564, 3.814, -33.549, -3.18]
  Call Extruder 0.0367
  MoveL (T18193) to (117.06, 119.45, 19.3) mm, rotated rx 180 ry 0 rz -180 deg; joints [2.107, 71.054, -37.564, 3.814, -33.549, -3.18]
  Call Extruder 0.26763
  MoveL (T18194) to (108.27, 119.45, 19.3) mm, rotated rx 180 ry 0 rz -180 deg; joints [2.046, 71.047, -37.551, 3.704, -33.551, -3.088]
  Call Extruder 0.08459
  MoveL (T18195) to (108.27, 116.67, 19.3) mm, rotated rx 180 ry 0 rz -180 deg; joints [2.046, 71.047, -37.551, 3.704, -33.551, -3.088]
  Call Extruder 0.14654
  MoveL (T18196) to (113.08, 116.67, 19.3) mm, rotated rx 180 ry 0 rz -180 deg; joints [2.479, 69.889, -35.374, 4.369, -34.592, -3.599]
  Call Extruder 0.32811
  MoveL (T18197) to (108.19, 107.08, 19.3) mm, rotated rx 180 ry 0 rz -180 deg; joints [2.479, 69.889, -35.374, 4.369, -34.592, -3.599]
  Call Extruder 0.03668
  MoveL (T18198) to (108.19, 105.88, 19.3) mm, rotated rx 180 ry 0 rz -180 deg; joints [2.418, 69.882, -35.361, 4.261, -34.595, -3.509]
  Call Extruder 0.02276
  MoveL (T18199) to (108.94, 105.88, 19.3) mm, rotated rx 180 ry 0 rz -180 deg; joints [2.418, 69.882, -35.361, 4.261, -34.595, -3.509]
  Set speed (150.0 mm/s)
  MoveL (T18200) to (108.6, 106.28, 19.3) mm, rotated rx 180 ry 0 rz -180 deg; joints [2.418, 69.882, -35.361, 4.261, -34.595, -3.509]
  Set speed (25.0 mm/s)
  MoveL (T18201) to (108.6, 106.28, 19.3) mm, rotated rx 180 ry 0 rz -180 deg; joints [1.985, 71.041, -37.539, 3.594, -33.554, -2.996]
  Call Extruder 0.25102
  MoveL (T18202) to (116.84, 106.28, 19.3) mm, rotated rx 180 ry 0 rz -180 deg; joints [1.985, 71.041, -37.539, 3.594, -33.554, -2.996]
  Call Extruder 0.05979
  MoveL (T18203) to (116.84, 108.25, 19.3) mm, rotated rx 180 ry 0 rz -180 deg; joints [1.925, 71.035, -37.528, 3.483, -33.556, -2.904]
  Call Extruder 0.16307
  MoveL (T18204) to (111.48, 108.25, 19.3) mm, rotated rx 180 ry 0 rz -180 deg; joints [1.925, 71.035, -37.528, 3.483, -33.556, -2.904]
  Call Extruder 0.3456
  MoveL (T18205) to (116.65, 118.34, 19.3) mm, rotated rx 180 ry 0 rz -180 deg; joints [1.925, 71.035, -37.528, 3.483, -33.556, -2.904]
  Call Extruder 0.02131
  MoveL (T18206) to (116.65, 119.04, 19.3) mm, rotated rx 180 ry 0 rz -180 deg; joints [2.356, 69.874, -35.348, 4.152, -34.597, -3.42]
  Call Extruder 0.24283
  MoveL (T18207) to (108.68, 119.04, 19.3) mm, rotated rx 180 ry 0 rz -180 deg; joints [2.295, 69.867, -35.334, 4.044, -34.6, -3.331]
  Call Extruder 0.05979
  MoveL (T18208) to (108.68, 117.08, 19.3) mm, rotated rx 180 ry 0 rz -180 deg; joints [2.295, 69.867, -35.334, 4.044, -34.6, -3.331]
  Call Extruder 0.15438
  MoveL (T18209) to (113.75, 117.08, 19.3) mm, rotated rx 180 ry 0 rz -180 deg; joints [1.864, 71.029, -37.516, 3.373, -33.558, -2.812]
  Call Extruder 0.34538
  MoveL (T18210) to (108.6, 106.98, 19.3) mm, rotated rx 180 ry 0 rz -180 deg; joints [1.864, 71.029, -37.516, 3.373, -33.558, -2.812]
  Call Extruder 0.01947
  MoveL (T18211) to (108.6, 106.34, 19.3) mm, rotated rx 180 ry 0 rz -180 deg; joints [1.83, 71.025, -37.51, 3.311, -33.559, -2.76]
  Set speed (150.0 mm/s)
  MoveL (T18212) to (108.54, 105.89, 19.3) mm, rotated rx 180 ry 0 rz -180 deg; joints [1.83, 71.025, -37.51, 3.311, -33.559, -2.76]
  Set speed (45.0 mm/s)
  Call Extruder -1.6
  MoveL (T18213) to (108.54, 105.89, 19.3) mm, rotated rx 180 ry 0 rz -180 deg; joints [1.83, 71.025, -37.51, 3.311, -33.559, -2.76]
  Set speed (120.0 mm/s)
  MoveL (T18214) to (108.54, 105.89, 19.3) mm, rotated rx 180 ry 0 rz -180 deg; joints [1.83, 70.946, -37.362, 3.307, -33.629, -2.754]
  Call Extruder -0.38
  MoveL (T18215) to (109.66, 106.33, 19.3) mm, rotated rx 180 ry 0 rz -180 deg; joints [1.83, 70.946, -37.362, 3.307, -33.629, -2.754]
  Set speed (45.0 mm/s)
  Call Extruder -0.02
  MoveL (T18216) to (109.66, 106.33, 19.3) mm, rotated rx 180 ry 0 rz -180 deg; joints [2.234, 69.861, -35.322, 3.936, -34.602, -3.242]
  Set speed (150.0 mm/s)
  MoveL (T18217) to (109.66, 106.33, 21.3) mm, rotated rx 180 ry 0 rz -180 deg; joints [2.234, 69.861, -35.322, 3.936, -34.602, -3.242]
  MoveL (T18218) to (104.34, 103.54, 21.3) mm, rotated rx 180 ry 0 rz -180 deg; joints [2.173, 69.854, -35.31, 3.828, -34.604, -3.152]
  MoveL (T18219) to (104.34, 103.54, 19.3) mm, rotated rx 180 ry 0 rz -180 deg; joints [2.173, 69.854, -35.31, 3.828, -34.604, -3.152]
  Set speed (40.0 mm/s)
  Call Extruder 2.0
  MoveL (T18220) to (104.34, 103.54, 19.3) mm, rotated rx 180 ry 0 rz -180 deg; joints [2.173, 69.854, -35.31, 3.828, -34.604, -3.152]
  Call Extruder 0.52159
  MoveL (T18221) to (121.46, 103.54, 19.3) mm, rotated rx 180 ry 0 rz -180 deg; joints [2.173, 69.854, -35.31, 3.828, -34.604, -3.152]
  Call Extruder 0.54596
